(* CoDeSys 2.3.9.41 project: henkel.pro *)
(* Libraries: TcpIp.lib 21.3.13 07:03:14, TcBase.lib 14.5.09 12:14:08, TcSystem.lib 27.2.12 15:08:36, TcBaseMath.lib 27.7.04 12:07:56, TcMath.lib 23.9.04 15:15:30, TcMC2.lib 10.7.13 15:31:24, STANDARD.LIB 5.6.98 12:03:02, TcNC.lib 10.10.08 18:55:34, TcUtilities.lib 10.1.13 20:12:12, SysLibTargetVisu.lib 16.6.08 16:24:26, SysLibVisu.lib 7.7.04 18:17:22 *)

(* Task configuration *)
TASK Standard (PRIORITY := 1, INTERVAL := T#5ms);
	MAIN
END_TASK
TASK Fast (PRIORITY := 0, INTERVAL := T#1ms);
	MainFast();
END_TASK

(* Global variable list: Globale_Variablen *)
VAR_GLOBAL
	trigger1  AT %Q*: BOOL;			(*to tigger the auduino pin 6 motor running*)
	trigger2  AT %Q*: BOOL;			(*to tigger the auduino pin 7* in velocity*)
	encoderX:	ARRAY[1..5] OF		LREAL;
	encoderY:	ARRAY[1..5] OF		LREAL;
	heading:		ARRAY[1..5] OF		LREAL;
	reset:		BOOL;
	home: BOOL;
	combinedX: LREAL;
	combinedY: LREAL;
	combinedH: LREAL;
(*for ROS*)
	robotPosX:	LREAL;
	robotPosY:	LREAL;
	robotPosTheta:	LREAL;
	robotVelX:	LREAL;
	robotVelY:	LREAL;
	robotVelTheta:	LREAL;
(*
###################
	TwinCAT NC Achsen
###################
*)


	Axis1 : AXIS_REF;
	PowerAxis1: MC_Power;
	MoveAxis1: MC_MoveVelocity;
	MoveAxis12: MC_MoveVelocity;
	ResetAxis1: MC_Reset;		(* debug function block output data *)
	HaltAxis1: MC_Halt;

	Axis2 : AXIS_REF;
	PowerAxis2: MC_Power;
	MoveAxis2: MC_MoveVelocity;
	MoveAxis22: MC_MoveVelocity;
	ResetAxis2: MC_Reset;		(* debug function block output data *)
	HaltAxis2: MC_Halt;

	Axis3 : AXIS_REF;
	PowerAxis3: MC_Power;
	MoveAxis3: MC_MoveVelocity;
	MoveAxis32: MC_MoveVelocity;
	ResetAxis3: MC_Reset;		(* debug function block output data *)
	HaltAxis3: MC_Halt;

	Axis4 : AXIS_REF;
	PowerAxis4: MC_Power;
	MoveAxis4: MC_MoveVelocity;
	MoveAxis42: MC_MoveVelocity;
	ResetAxis4: MC_Reset;		(* debug function block output data *)
	HaltAxis4: MC_Halt;
END_VAR

(* Global variable list: TwinCAT_Configuration *)
(* Generated automatically by TwinCAT - (read only) *)
VAR_CONFIG
	MainFast.fblocalization.encoder1.PlcToNc AT %QB1156 : PLCTONC_AXIS_REF;
	MainFast.fblocalization.encoder1.NcToPlc AT %IB1152 : NCTOPLC_AXIS_REF;
	MainFast.fblocalization.encoder2.PlcToNc AT %QB1284 : PLCTONC_AXIS_REF;
	MainFast.fblocalization.encoder2.NcToPlc AT %IB1280 : NCTOPLC_AXIS_REF;
	MainFast.fblocalization.encoder3.PlcToNc AT %QB1412 : PLCTONC_AXIS_REF;
	MainFast.fblocalization.encoder3.NcToPlc AT %IB1408 : NCTOPLC_AXIS_REF;
	MainFast.fblocalization.encoder4.PlcToNc AT %QB1540 : PLCTONC_AXIS_REF;
	MainFast.fblocalization.encoder4.NcToPlc AT %IB1536 : NCTOPLC_AXIS_REF;
	.trigger1 AT %QX1152.0 : BOOL;
	.trigger2 AT %QX1152.1 : BOOL;
END_VAR

(* Global variable list: Variablen_Konfiguration *)
VAR_CONFIG
	Axis1.PlcToNc AT %QB128 : PLCTONC_AXIS_REF;	(*  ~ {LinkedWith:TINC^NC-Task 1 SAF^Achsen^Achse 1^Eingänge^Achse 1_FromPlc} *)
	Axis1.NcToPlc AT %IB128 : NCTOPLC_AXIS_REF;	(*  ~ {LinkedWith:TINC^NC-Task 1 SAF^Achsen^Achse 1^Ausgänge^Achse 1_ToPlc} *)
	Axis2.PlcToNc AT %QB256 : PLCTONC_AXIS_REF;	(*  ~ {LinkedWith:TINC^NC-Task 1 SAF^Achsen^Achse 2^Eingänge^Achse 2_FromPlc} *)
	Axis2.NcToPlc AT %IB256 : NCTOPLC_AXIS_REF;	(*  ~ {LinkedWith:TINC^NC-Task 1 SAF^Achsen^Achse 2^Ausgänge^Achse 2_ToPlc} *)
	Axis3.PlcToNc AT %QB512 : PLCTONC_AXIS_REF;
	Axis3.NcToPlc AT %IB512 : NCTOPLC_AXIS_REF;
	Axis4.PlcToNc AT %QB1024 : PLCTONC_AXIS_REF;
	Axis4.NcToPlc AT %IB1024 : NCTOPLC_AXIS_REF;
END_VAR

(* Data type *)
TYPE MoveState_NC :
(
	NC_INIT,
	NC_ENABLE,
	NC_MOVE,
	NC_MOVENEXT,
	NC_ERROR,
	NC_RESET
);
END_TYPE

(* POU MAIN, ST *)
PROGRAM MAIN
VAR
	fbPLC_Reset:  PLC_Reset;
	fbPLC_Start:  PLC_Start;
	state_NC : MoveState_NC;
(* manual runnning*)
	Manual: BOOL:=FALSE;
	bEnable: 			BOOL;										(* gibt die Achse frei *)
	bReset_Axis: 			BOOL;										(* Reset der Achse *)
	bAxis_Ready:		ARRAY[1..5] OF	BOOL;						(* Checks whether the axis is ready *)
	bMoveCombination:	ARRAY[1..10] OF		BOOL;					(*the combined movement*)
	i: INT;
	MotionReq: BOOL;
	timeToMove: TIME;
	directionToMove: INT;
	timeToMoveReal: LREAL;
	speedToMove:LREAL:=603;
	timeUp: BOOL;
	timerOn: BOOL;
	fbTON1: TON;



(*
###################
ROS TCP/IP CONNECTION
###################
*)
	myROS_connect_receiveData:				ROS_connect_receiveData;
	myROS_connect_sendData:				ROS_connect_sendData;
	myROS_disconnect:			ROS_disconnect;
	myROS_receiveData:			ROS_receiveData;
	myROS_sendData:			ROS_sendData;
	myROS_convertSendData:		ROS_convertSendData;

	ROS_tcpSocketReceiveData: T_HSOCKET;
	ROS_connectionOpenReceiveData: BOOL:=FALSE;

	ROS_tcpSocketSendData: T_HSOCKET;
	ROS_connectionOpenSendData: BOOL:=FALSE;

	ROS_closeConnection: BOOL:=TRUE;

	ROS_velAxis1: LREAL := 0;
	ROS_velAxis2: LREAL := 0;
	ROS_velAxis3: LREAL := 0;
	ROS_velAxis4: LREAL := 0;

	ROS_RobotPosX: LREAL := 0;
	ROS_RobotPosY: LREAL := 0;
	ROS_RobotPosTheta: LREAL:= 0;
	ROS_RobotVelX: LREAL:= 0;
	ROS_RobotVelY: LREAL:= 0;
	ROS_RobotVelTheta: LREAL:= 0;

	sendBufferREAL: LREAL:=0;
	sendBuffer: STRING;
	sendTakt: LREAL := 0;
	(*#END# ROS variables*)



	vel_last1 : LREAL;
	vel_current1 : LREAL;
	vel_last2 : LREAL;
	vel_current2 : LREAL;
	vel_last3 : LREAL;
	vel_current3 : LREAL;
	vel_last4 : LREAL;
	vel_current4 : LREAL;

(*
###################
ODOMETRY
###################
*)



	startTimer1: BOOL;
	timer1On: BOOL;

	firstStart: BOOL;
	Q: BOOL;
	startPLC: BOOL;
	oldSpeedX: LREAL;
	oldSpeedY: LREAL;
	oldSpeedH: LREAL;

(*JOSTICK*)
	connectJs:			jsConnect;
	disconnectJs:			jsDisconnect;
	receiveJsData:				jsReceiveData;
	tcpSockeJst: T_HSOCKET;
	connectionOpen_js: BOOL:=FALSE;
	closeConnection_js: BOOL:=TRUE;
	XAxis: LREAL;
	YAxis: LREAL;
	ZAxis: LREAL;
	botton: LREAL;

	myWP_tcpSocket: T_HSOCKET;
	myWP_connect:		WP_connect;
	myWP_disconnect:	WP_Disconnect;
	myWP_receiveData:	WP_ReceiveData;
	myWP_connected: BOOL := FALSE;
	myWP_connectionClosed: BOOL:=TRUE;
	wpBotton: LREAL;
END_VAR
(*
##
## This code was built by Theng Chua and Christian Scheifele, University of Stuttgart, 2014.
## It contains complete segments from Chris Jarrett, Auckland University, 2014
## and is derived in part from the TCP/IP server example on www.beckhoff.com
##
*)

(*
###################
Manual
###################
*)
IF (Manual=TRUE) THEN
	IF (reset=TRUE) THEN
	trigger1:=FALSE;
	trigger2:=TRUE;
	fbPLC_Reset(port:=801,RESET:=TRUE);
	fbPLC_Start(port:=801,start:=TRUE);
	reset:=FALSE;
	trigger1:=FALSE;
	trigger2:=FALSE;
	END_IF

	FOR i:=1 TO 10 BY 1 DO
		IF(bMoveCombination[i]) THEN
			directionToMove:=i;
			MotionReq:=TRUE;
		END_IF
	END_FOR

	IF(MotionReq=TRUE) THEN
		CASE directionToMove OF
		1:	ROS_velAxis1:= -speedToMove;
			ROS_velAxis2:= 0;
			ROS_velAxis3:= 0;
			ROS_velAxis4:= -speedToMove;
		2:	ROS_velAxis1:= -speedToMove;
			ROS_velAxis2:= -speedToMove;
			ROS_velAxis3:= -speedToMove;
			ROS_velAxis4:= -speedToMove;
		3:	ROS_velAxis1:= 0;
			ROS_velAxis2:= -speedToMove;
			ROS_velAxis3:= -speedToMove;
			ROS_velAxis4:= 0;
		4:	ROS_velAxis1:= -speedToMove;
			ROS_velAxis2:= speedToMove;
			ROS_velAxis3:= speedToMove;
			ROS_velAxis4:= -speedToMove;
		5:	ROS_velAxis1:= speedToMove;
			ROS_velAxis2:= -speedToMove;
			ROS_velAxis3:= -speedToMove;
			ROS_velAxis4:= speedToMove;
		6:	ROS_velAxis1:= 0;
			ROS_velAxis2:= speedToMove;
			ROS_velAxis3:= speedToMove;
			ROS_velAxis4:= 0;
		7:	ROS_velAxis1:= speedToMove;
			ROS_velAxis2:= speedToMove;
			ROS_velAxis3:= speedToMove;
			ROS_velAxis4:= speedToMove;
		8:	ROS_velAxis1:= speedToMove;
			ROS_velAxis2:= 0;
			ROS_velAxis3:= 0;
			ROS_velAxis4:= speedToMove;
		9:	ROS_velAxis1:= -speedToMove;
			ROS_velAxis2:= speedToMove;
			ROS_velAxis3:= -speedToMove;
			ROS_velAxis4:= speedToMove;
		10:	ROS_velAxis1:= speedToMove;
			ROS_velAxis2:= -speedToMove;
			ROS_velAxis3:= speedToMove;
			ROS_velAxis4:= -speedToMove;
		ELSE
			ROS_velAxis1:= 0;
			ROS_velAxis2:= 0;
			ROS_velAxis3:= 0;
			ROS_velAxis4:= 0;
		END_CASE
	timetomove:= REAL_TO_TIME (timeToMoveReal);
	timerOn:=TRUE;
	END_IF

	fbTON1(IN:=timerOn, PT:=timeToMove, Q=>timeUp, ET=>);

	IF (timeUp=TRUE)  THEN
	MotionReq:=FALSE;
	bMoveCombination[directionToMove]:=FALSE;
	ROS_velAxis1:= 0;
	ROS_velAxis2:= 0;
	ROS_velAxis3:= 0;
	ROS_velAxis4:= 0;
	directionToMove:=0;
	timerOn:=FALSE;
	END_IF
(*
###################
ODOMETRY
###################
*)

	IF (vel_current1<>0 OR vel_current2<>0 OR vel_current3<>0 OR vel_current4<>0) THEN trigger1:=TRUE;
	ELSE trigger1:=FALSE;
	END_IF

	trigger2:=(MoveAxis1.InVelocity AND MoveAxis2.InVelocity AND MoveAxis3.InVelocity AND MoveAxis4.InVelocity) OR (MoveAxis12.InVelocity AND MoveAxis22.InVelocity AND MoveAxis32.InVelocity AND MoveAxis42.InVelocity);

ELSE
(*
###################
ROS TCP/IP CONNECTION
###################

Close TCP port from last time-remove after DEBUG
	
		IF ROS_closeConnection THEN
		myROS_disconnect(bCloseAll:=ROS_closeConnection);
		ROS_closeConnection:=FALSE;
		END_IF*)

		(*Open a connection to ROS - Receive Data*)
		IF NOT ROS_connectionOpenReceiveData THEN
		myROS_connect_receiveData(RosConnected=>ROS_connectionOpenReceiveData, socketToUse=>ROS_tcpSocketReceiveData);
		END_IF
		IF ROS_connectionOpenReceiveData THEN
		myROS_receiveData(socketToUse:=ROS_tcpSocketReceiveData,velAxis1=>ROS_velAxis1, velAxis2=>ROS_velAxis2, velAxis3=>ROS_velAxis3, velAxis4=>ROS_velAxis4);
		END_IF

		(*Open a connection to ROS - Send Data*)
		IF NOT ROS_connectionOpenSendData THEN
		myROS_connect_sendData(RosConnected=>ROS_connectionOpenSendData, socketToUse=>ROS_tcpSocketSendData);
		END_IF

		(*ODOMETRY SORCE*)
		ROS_RobotPosX := robotPosY;
		ROS_RobotPosY := robotPosX;
		ROS_RobotPosTheta := robotPosTheta;
		ROS_RobotVelX := RobotVelY;
		ROS_RobotVelY := RobotVelX;
		ROS_RobotVelTheta := RobotVelTheta;

		IF ROS_connectionOpenSendData THEN
		(* TAKTZEIT EINSTELLEN *)
		sendTakt := sendTakt + 0.1;
			IF sendTakt > 1THEN
			myROS_convertSendData(robotPosX:=ROS_RobotPosX, robotPosY:=ROS_RobotPosY, robotPosTheta:= ROS_RobotPosTheta, robotVelX:=ROS_RobotVelX, robotVelY:=ROS_RobotVelY, robotVelTheta:=ROS_RobotVelTheta, send_message=>sendBuffer );
			myROS_sendData(sendBuffer:=sendBuffer, socketToUse:=ROS_tcpSocketSendData);
			sendTakt := 0;
			END_IF
		END_IF



	(*JOSTICK*)
	(*Close TCP port from last time-remove after DEBUG*)
	IF closeConnection_js THEN
	disconnectJs(bCloseAll:=closeConnection_js);
	closeConnection_js:=FALSE;
	END_IF

	(*Open a connection*)
	IF (connectionOpen_js=FALSE) THEN
	connectJs(arduinoConnected=>connectionOpen_js, socketToUse=>tcpSockeJst);
	END_IF

	IF (connectionOpen_js=TRUE) THEN
	receiveJsData(socketToUse:=tcpSockeJst ,botton=>botton, xAxis=>XAxis, yAxis=>YAxis, zAxis=>ZAxis);
	END_IF

	(*IF  (botton = 48 OR botton = 32) THEN
	ROS_velAxis1:= -YAxis+XAxis-ZAxis;
	ROS_velAxis2:= -YAxis-XAxis+ZAxis;
	ROS_velAxis3:= -YAxis-XAxis-ZAxis;
	ROS_velAxis4:= -YAxis+XAxis+ZAxis;
	ELSE
	ROS_velAxis1:= 0;
	ROS_velAxis2:= 0;
	ROS_velAxis3:= 0;
	ROS_velAxis4:= 0;
	END_IF*)

(*Windows Phone Connection*)

	IF (myWP_connectionClosed) THEN
	myWP_disconnect(bCloseAll:=myWP_connectionClosed);
	myWP_connectionClosed:=FALSE;
	END_IF

	IF (myWP_connected=FALSE) THEN
	myWP_connect(WPConnected=>myWP_connected, socketToUse=>myWP_tcpSocket);
	END_IF

	IF (myWP_connected=TRUE) THEN
	myWP_receiveData(socketToUse:=myWP_tcpSocket ,botton=>wpBotton, xAxis=>XAxis, yAxis=>YAxis, zAxis=>ZAxis);
		(*IF(wpBotton <> 0 ) THEN
			ROS_velAxis1:= -YAxis+XAxis-ZAxis;
			ROS_velAxis2:= -YAxis-XAxis+ZAxis;
			ROS_velAxis3:= -YAxis-XAxis-ZAxis;
			ROS_velAxis4:= -YAxis+XAxis+ZAxis;
		END_IF*)
		wpBotton := 0;
	END_IF

END_IF (* for manual running*)

(*
###################
TwinCAT NC Achsen
###################
*)
Axis1.ReadStatus;
Axis2.ReadStatus;
Axis3.ReadStatus;
Axis4.ReadStatus;

vel_current1 := -ROS_velAxis1;
vel_current2 := ROS_velAxis2;
vel_current3 := -ROS_velAxis3;
vel_current4 := ROS_velAxis4;

(* move axis using a state machine *)
CASE state_NC OF
		NC_INIT :	(* initialisation *)
			(* initialize all function blocks *)
			MoveAxis1.Execute := FALSE;
			ResetAxis1.Execute := FALSE;
			MoveAxis2.Execute := FALSE;
			ResetAxis2.Execute := FALSE;
			MoveAxis3.Execute := FALSE;
			ResetAxis3.Execute := FALSE;
			MoveAxis4.Execute := FALSE;
			ResetAxis4.Execute := FALSE;
			MoveAxis12.Execute := FALSE;
			MoveAxis22.Execute := FALSE;
			MoveAxis32.Execute := FALSE;
			MoveAxis42.Execute := FALSE;
			HaltAxis1.Execute := FALSE;
			HaltAxis2.Execute := FALSE;
			HaltAxis3.Execute := FALSE;
			HaltAxis4.Execute := FALSE;

			state_NC := NC_ENABLE;

		NC_ENABLE :
			PowerAxis1.Enable := TRUE;
			PowerAxis1.Enable_Positive := TRUE;
			PowerAxis1.Enable_Negative := TRUE;
			PowerAxis2.Enable := TRUE;
			PowerAxis2.Enable_Positive := TRUE;
			PowerAxis2.Enable_Negative := TRUE;
			PowerAxis3.Enable := TRUE;
			PowerAxis3.Enable_Positive := TRUE;
			PowerAxis3.Enable_Negative := TRUE;
			PowerAxis4.Enable := TRUE;
			PowerAxis4.Enable_Positive := TRUE;
			PowerAxis4.Enable_Negative := TRUE;

			IF PowerAxis1.Status AND PowerAxis2.Status AND PowerAxis3.Status AND PowerAxis4.Status THEN
				state_NC := NC_MOVE;
			ELSIF PowerAxis1.Error AND PowerAxis2.Error AND PowerAxis3.Error AND PowerAxis4.Error THEN
				state_NC := NC_ERROR;
			END_IF

		NC_MOVE :
			IF vel_current1>0 THEN
				HaltAxis1.Execute := FALSE;
				MoveAxis1.Direction := MC_Positive_Direction;
				MoveAxis1.Velocity := vel_current1;
				MoveAxis1.BufferMode := MC_Aborting;
				MoveAxis1.Execute := TRUE;
			ELSIF vel_current1<0 THEN
				HaltAxis1.Execute := FALSE;
				MoveAxis1.Direction := MC_Negative_Direction;
				MoveAxis1.Velocity := -vel_current1;
				MoveAxis1.BufferMode := MC_Aborting;
				MoveAxis1.Execute := TRUE;
			ELSE
				HaltAxis1.BufferMode := MC_Aborting;
				HaltAxis1.Execute := TRUE;
			END_IF;


			IF vel_current2>0 THEN
				HaltAxis2.Execute := FALSE;
				MoveAxis2.Direction := MC_Positive_Direction;
				MoveAxis2.Velocity := vel_current2;
				MoveAxis2.BufferMode := MC_Aborting;
				MoveAxis2.Execute := TRUE;
			ELSIF vel_current2<0 THEN
				HaltAxis2.Execute := FALSE;
				MoveAxis2.Direction := MC_Negative_Direction;
				MoveAxis2.Velocity := -vel_current2;
				MoveAxis2.BufferMode := MC_Aborting;
				MoveAxis2.Execute := TRUE;
			ELSE
				HaltAxis2.BufferMode := MC_Aborting;
				HaltAxis2.Execute := TRUE;
			END_IF;


			IF vel_current3>0 THEN
				HaltAxis3.Execute := FALSE;
				MoveAxis3.Direction := MC_Positive_Direction;
				MoveAxis3.Velocity := vel_current3;
				MoveAxis3.BufferMode := MC_Aborting;
				MoveAxis3.Execute := TRUE;
			ELSIF vel_current3<0 THEN
				HaltAxis3.Execute := FALSE;
				MoveAxis3.Direction := MC_Negative_Direction;
				MoveAxis3.Velocity := -vel_current3;
				MoveAxis3.BufferMode := MC_Aborting;
				MoveAxis3.Execute := TRUE;
			ELSE
				HaltAxis3.BufferMode := MC_Aborting;
				HaltAxis3.Execute := TRUE;
			END_IF;


			IF vel_current4>0 THEN
				HaltAxis4.Execute := FALSE;
				MoveAxis4.Direction := MC_Positive_Direction;
				MoveAxis4.Velocity := vel_current4;
				MoveAxis4.BufferMode := MC_Aborting;
				MoveAxis4.Execute := TRUE;
			ELSIF vel_current4<0 THEN
				HaltAxis4.Execute := FALSE;
				MoveAxis4.Direction := MC_Negative_Direction;
				MoveAxis4.Velocity := -vel_current4;
				MoveAxis4.BufferMode := MC_Aborting;
				MoveAxis4.Execute := TRUE;
			ELSE
				HaltAxis4.BufferMode := MC_Aborting;
				HaltAxis4.Execute := TRUE;
			END_IF;

			IF vel_last1<>vel_current1 OR vel_last2<>vel_current2 OR vel_last3<>vel_current3 OR vel_last4<>vel_current4 THEN
				MoveAxis1.Execute := FALSE;
				MoveAxis2.Execute := FALSE;
				MoveAxis3.Execute := FALSE;
				MoveAxis4.Execute := FALSE;
				vel_last1 := vel_current1;
				vel_last2 := vel_current2;
				vel_last3 := vel_current3;
				vel_last4 := vel_current4;
				state_NC := NC_MOVENEXT;
			END_IF;
			IF  MoveAxis1.CommandAborted OR MoveAxis1.Error OR MoveAxis2.CommandAborted OR MoveAxis2.Error OR MoveAxis3.CommandAborted OR MoveAxis3.Error OR MoveAxis4.CommandAborted OR MoveAxis4.Error THEN
				state_NC := NC_MOVE;
			END_IF

		NC_MOVENEXT :
			IF vel_current1>0 THEN
				HaltAxis1.Execute := FALSE;
				MoveAxis12.Direction := MC_Positive_Direction;
				MoveAxis12.Velocity := vel_current1;
				MoveAxis12.BufferMode := MC_Aborting;
				MoveAxis12.Execute := TRUE;
			ELSIF vel_current1<0 THEN
				HaltAxis1.Execute := FALSE;
				MoveAxis12.Direction := MC_Negative_Direction;
				MoveAxis12.Velocity := -vel_current1;
				MoveAxis12.BufferMode := MC_Aborting;
				MoveAxis12.Execute := TRUE;
			ELSE
				HaltAxis1.BufferMode := MC_Aborting;
				HaltAxis1.Execute := TRUE;
			END_IF;


			IF vel_current2>0 THEN
				HaltAxis2.Execute := FALSE;
				MoveAxis22.Direction := MC_Positive_Direction;
				MoveAxis22.Velocity := vel_current2;
				MoveAxis22.BufferMode := MC_Aborting;
				MoveAxis22.Execute := TRUE;
			ELSIF vel_current2<0 THEN
				HaltAxis2.Execute := FALSE;
				MoveAxis22.Direction := MC_Negative_Direction;
				MoveAxis22.Velocity := -vel_current2;
				MoveAxis22.BufferMode := MC_Aborting;
				MoveAxis22.Execute := TRUE;
			ELSE
				HaltAxis2.BufferMode := MC_Aborting;
				HaltAxis2.Execute := TRUE;
			END_IF;


			IF vel_current3>0 THEN
				HaltAxis3.Execute := FALSE;
				MoveAxis32.Direction := MC_Positive_Direction;
				MoveAxis32.Velocity := vel_current3;
				MoveAxis32.BufferMode := MC_Aborting;
				MoveAxis32.Execute := TRUE;
			ELSIF vel_current3<0 THEN
				HaltAxis3.Execute := FALSE;
				MoveAxis32.Direction := MC_Negative_Direction;
				MoveAxis32.Velocity := -vel_current3;
				MoveAxis32.BufferMode := MC_Aborting;
				MoveAxis32.Execute := TRUE;
			ELSE
				HaltAxis3.BufferMode := MC_Aborting;
				HaltAxis3.Execute := TRUE;
			END_IF;


			IF vel_current4>0 THEN
				HaltAxis4.Execute := FALSE;
				MoveAxis42.Direction := MC_Positive_Direction;
				MoveAxis42.Velocity := vel_current4;
				MoveAxis42.BufferMode := MC_Aborting;
				MoveAxis42.Execute := TRUE;
			ELSIF vel_current4<0 THEN
				HaltAxis4.Execute := FALSE;
				MoveAxis42.Direction := MC_Negative_Direction;
				MoveAxis42.Velocity := -vel_current4;
				MoveAxis42.BufferMode := MC_Aborting;
				MoveAxis42.Execute := TRUE;
			ELSE
				HaltAxis4.BufferMode := MC_Aborting;
				HaltAxis4.Execute := TRUE;
			END_IF;

			IF vel_last1<>vel_current1 OR vel_last2<>vel_current2 OR vel_last3<>vel_current3 OR vel_last4<>vel_current4 THEN
				MoveAxis12.Execute := FALSE;
				MoveAxis22.Execute := FALSE;
				MoveAxis32.Execute := FALSE;
				MoveAxis42.Execute := FALSE;
				vel_last1 := vel_current1;
				vel_last2 := vel_current2;
				vel_last3 := vel_current3;
				vel_last4 := vel_current4;
				state_NC := NC_MOVE;
			END_IF;
			IF  MoveAxis12.CommandAborted OR MoveAxis12.Error OR MoveAxis22.CommandAborted OR MoveAxis22.Error OR MoveAxis32.CommandAborted OR MoveAxis32.Error OR MoveAxis42.CommandAborted OR MoveAxis42.Error THEN
				state_NC := NC_MOVE;
			END_IF


		NC_ERROR :
			IF Axis1.Status.Error OR Axis2.Status.Error OR Axis3.Status.Error OR Axis4.Status.Error THEN
				state_NC := NC_RESET;	(* axis error requires reset *)
			ELSE
				state_NC := NC_INIT;		(* function block errors don't need a reset *)
			END_IF

		NC_RESET :
			ResetAxis1.Execute := TRUE;
			ResetAxis2.Execute := TRUE;
			ResetAxis3.Execute := TRUE;
			ResetAxis4.Execute := TRUE;
			IF ResetAxis1.Done AND ResetAxis2.Done AND ResetAxis3.Done AND ResetAxis4.Done THEN
				state_NC := NC_INIT;
			ELSIF ResetAxis1.Error OR ResetAxis2.Error OR ResetAxis3.Error OR ResetAxis4.Error THEN
				state_NC := NC_INIT; (* can't do anything here *)
			END_IF

END_CASE

ActPower;	(* call the power function block *)
ActMove;	(* call the move function block *)
ActReset;	(* call the reset function block *)
ActHaltAxis1;
ActHaltAxis2;
ActHaltAxis3;
ActHaltAxis4;
END_PROGRAM
ACTION ActHaltAxis1:
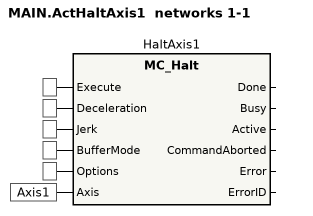
_FBD_ (* Function Block Diagram *)
NETWORK 1
	HaltAxis1:MC_Halt(Execute: , Deceleration: , Jerk: , BufferMode: , Options: , Axis: Axis1)
_END_FBD_
END_ACTION
ACTION ActHaltAxis2:
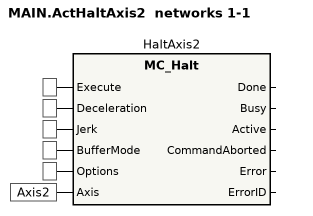
_FBD_ (* Function Block Diagram *)
NETWORK 1
	HaltAxis2:MC_Halt(Execute: , Deceleration: , Jerk: , BufferMode: , Options: , Axis: Axis2)
_END_FBD_
END_ACTION
ACTION ActHaltAxis3:
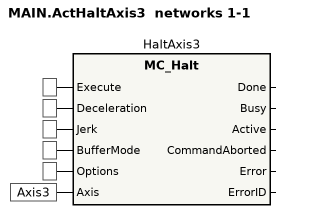
_FBD_ (* Function Block Diagram *)
NETWORK 1
	HaltAxis3:MC_Halt(Execute: , Deceleration: , Jerk: , BufferMode: , Options: , Axis: Axis3)
_END_FBD_
END_ACTION
ACTION ActHaltAxis4:
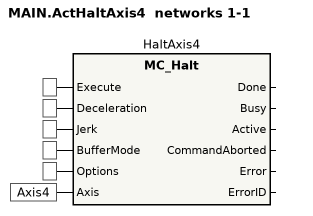
_FBD_ (* Function Block Diagram *)
NETWORK 1
	HaltAxis4:MC_Halt(Execute: , Deceleration: , Jerk: , BufferMode: , Options: , Axis: Axis4)
_END_FBD_
END_ACTION
ACTION ActMove:
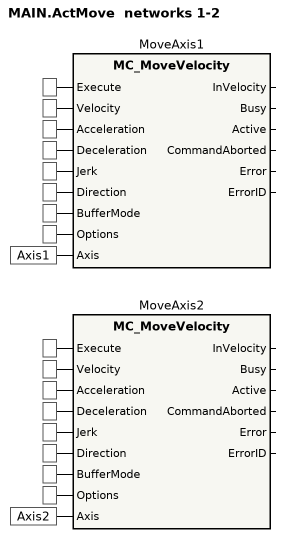
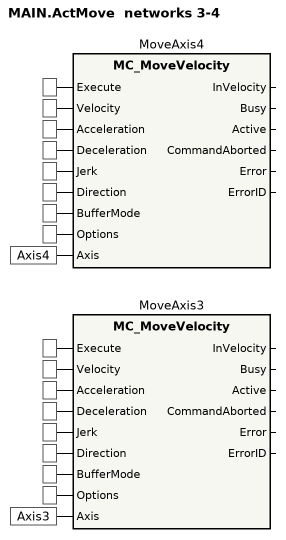
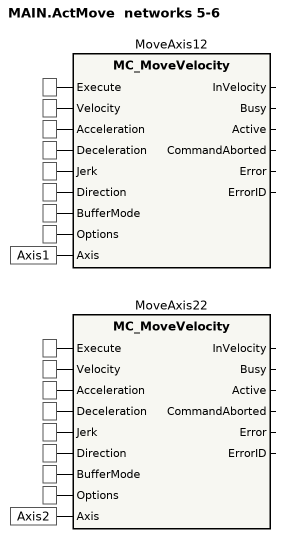
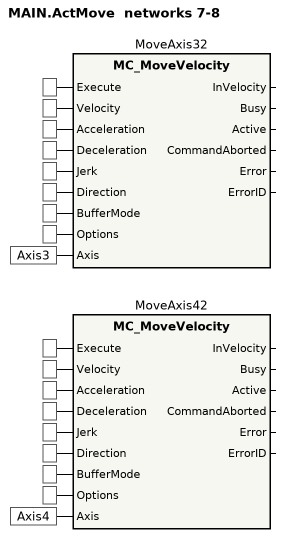
_FBD_ (* Function Block Diagram *)
NETWORK 1
	MoveAxis1:MC_MoveVelocity(Execute: , Velocity: , Acceleration: , Deceleration: , Jerk: , Direction: , BufferMode: , Options: , Axis: Axis1)
NETWORK 2
	MoveAxis2:MC_MoveVelocity(Execute: , Velocity: , Acceleration: , Deceleration: , Jerk: , Direction: , BufferMode: , Options: , Axis: Axis2)
NETWORK 3
	MoveAxis4:MC_MoveVelocity(Execute: , Velocity: , Acceleration: , Deceleration: , Jerk: , Direction: , BufferMode: , Options: , Axis: Axis4)
NETWORK 4
	MoveAxis3:MC_MoveVelocity(Execute: , Velocity: , Acceleration: , Deceleration: , Jerk: , Direction: , BufferMode: , Options: , Axis: Axis3)
NETWORK 5
	MoveAxis12:MC_MoveVelocity(Execute: , Velocity: , Acceleration: , Deceleration: , Jerk: , Direction: , BufferMode: , Options: , Axis: Axis1)
NETWORK 6
	MoveAxis22:MC_MoveVelocity(Execute: , Velocity: , Acceleration: , Deceleration: , Jerk: , Direction: , BufferMode: , Options: , Axis: Axis2)
NETWORK 7
	MoveAxis32:MC_MoveVelocity(Execute: , Velocity: , Acceleration: , Deceleration: , Jerk: , Direction: , BufferMode: , Options: , Axis: Axis3)
NETWORK 8
	MoveAxis42:MC_MoveVelocity(Execute: , Velocity: , Acceleration: , Deceleration: , Jerk: , Direction: , BufferMode: , Options: , Axis: Axis4)
_END_FBD_
END_ACTION
ACTION ActPower:
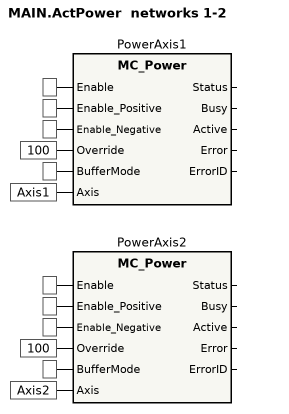
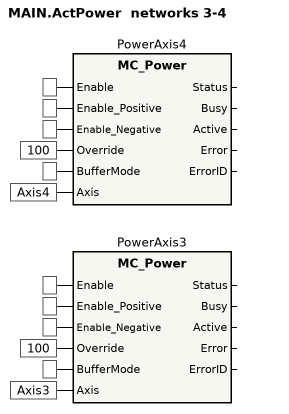
_FBD_ (* Function Block Diagram *)
NETWORK 1
	PowerAxis1:MC_Power(Enable: , Enable_Positive: , Enable_Negative: , Override: 100, BufferMode: , Axis: Axis1)
NETWORK 2
	PowerAxis2:MC_Power(Enable: , Enable_Positive: , Enable_Negative: , Override: 100, BufferMode: , Axis: Axis2)
NETWORK 3
	PowerAxis4:MC_Power(Enable: , Enable_Positive: , Enable_Negative: , Override: 100, BufferMode: , Axis: Axis4)
NETWORK 4
	PowerAxis3:MC_Power(Enable: , Enable_Positive: , Enable_Negative: , Override: 100, BufferMode: , Axis: Axis3)
_END_FBD_
END_ACTION
ACTION ActReset:
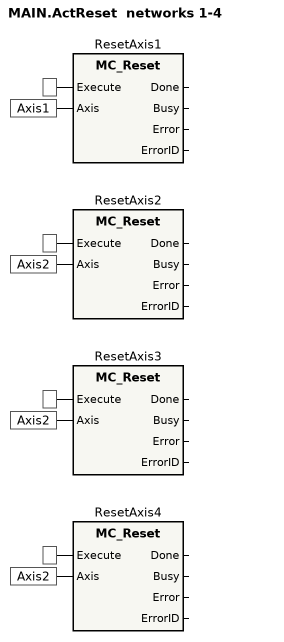
_FBD_ (* Function Block Diagram *)
NETWORK 1
	ResetAxis1:MC_Reset(Execute: , Axis: Axis1)
NETWORK 2
	ResetAxis2:MC_Reset(Execute: , Axis: Axis2)
NETWORK 3
	ResetAxis3:MC_Reset(Execute: , Axis: Axis2)
NETWORK 4
	ResetAxis4:MC_Reset(Execute: , Axis: Axis2)
_END_FBD_
END_ACTION

(* POU ROS_connect_receiveData, ST *)
FUNCTION_BLOCK ROS_connect_receiveData
VAR


	(*Functions*)
	openSocket: BOOL:=FALSE;
	fb_listen: FB_SocketListen;
	fb_accept: FB_SocketAccept;
	(*Timers*)
	fbAcceptTON: TON;

	(*TCP socket variables*)
	activeSocketHandle: T_HSOCKET;
	socketHandle: T_HSOCKET;



	(*Error variables*)
	listenError: UDINT:=0;
	acceptError: UDINT;
	listenErrSet: BOOL;
	closeError: UDINT;
	sendError: UDINT;
	receiveError: UDINT;
	bSendError: BOOL;


	(*Trigger Variables*)
	bCloseAll: BOOL := TRUE;

	(*Connection information*)
	portNumber: INT:=711;
	bAccepted: BOOL;

	(*Constants*)
	PLCPRJ_ACCEPT_POLLING_TIME: TIME:=T#1s;

	display: LREAL;
	heading: LREAL;

	state: INT:=0;

	xDist: LREAL;
	yDist: LREAL;
	zDist: LREAL;


	listening: BOOL;
END_VAR
VAR_OUTPUT
	RosConnected: BOOL;
	socketToUse: T_HSOCKET;
END_VAR
(*
##
## This code was built by Christian Scheifele, University of Stuttgart, 2014.
## It contains complete segments from Chris Jarrett, Auckland University, 2014
## and is derived in part from the TCP/IP server example on www.beckhoff.com
##
*)

CASE state OF
0:

IF(fb_Listen.hListener.localAddr.nPort=portNumber) THEN
RETURN;

ELSE
state:=1;
END_IF

1:
fb_listen
(
	sSrvNetId:='' ,
	sLocalHost:='',
	nLocalPort:=portNumber,
	bExecute:=TRUE,
	tTimeout:=T#5s,
	hListener=>socketHandle,
	nErrId=>listenError,
	bError=>listenErrSet,

);

	IF(fb_Listen.hListener.localAddr.nPort=portNumber) THEN
		fb_listen(bExecute:=FALSE); 		(*Start listening and move to the accept state*)

		state:=2;
	ELSE
		(*Return to the listening state*)
		state:=1;
	END_IF



2:

(*Start accepting a client connection*)
fbAcceptTON( IN := TRUE, PT := T#2s);  (*Start a timer to poll for the accepted connection*)
		IF fbAcceptTON.Q THEN
			fbAcceptTON( IN := FALSE );	(*Reset timer*)
			fb_accept(  bExecute := FALSE  ); (*Generate a rising edge to activate the accept function*)
			fb_accept(hListener := socketHandle, bExecute:= TRUE, hSocket=>activeSocketHandle );
			state:=3; (*Move to the state where the client is accepted*)

			fbAcceptTON( IN := FALSE);

		END_IF
3:
(*Complete accpeting the client connection*)
	fb_accept( bExecute := FALSE ); (*Reset the accept function to try connection again if necessary*)
	IF NOT fb_accept.bBusy THEN
		IF NOT fb_accept.bError THEN
			IF fb_accept.bAccepted THEN
				bAccepted := TRUE; (*If the client connection is accepted without error then move to the send state*)
				fb_accept(bExecute:=FALSE);
				socketToUse:=fb_accept.hSocket;
				state:=4;
			ELSE
				fb_listen(bExecute:=FALSE);
				fb_accept(bExecute:=FALSE);
				RosConnected:=FALSE; (*If the connection attempt was not successful, return the boolean as false*)
				fbAcceptTON( IN := FALSE);
				state:=2;
			END_IF
		END_IF
	END_IF
4:
RosConnected:=TRUE;
RETURN;

END_CASE;
END_FUNCTION_BLOCK

(* POU ROS_connect_sendData, ST *)
FUNCTION_BLOCK ROS_connect_sendData
VAR


	(*Functions*)
	openSocket: BOOL:=FALSE;
	fb_listen: FB_SocketListen;
	fb_accept: FB_SocketAccept;
	(*Timers*)
	fbAcceptTON: TON;

	(*TCP socket variables*)
	activeSocketHandle: T_HSOCKET;
	socketHandle: T_HSOCKET;



	(*Error variables*)
	listenError: UDINT:=0;
	acceptError: UDINT;
	listenErrSet: BOOL;
	closeError: UDINT;
	sendError: UDINT;
	receiveError: UDINT;
	bSendError: BOOL;


	(*Trigger Variables*)
	bCloseAll: BOOL := TRUE;

	(*Connection information*)
	portNumber: INT:=712;
	bAccepted: BOOL;

	(*Constants*)
	PLCPRJ_ACCEPT_POLLING_TIME: TIME:=T#1s;

	display: LREAL;
	heading: LREAL;

	state: INT:=0;

	xDist: LREAL;
	yDist: LREAL;
	zDist: LREAL;


	listening: BOOL;
END_VAR
VAR_OUTPUT
	RosConnected: BOOL;
	socketToUse: T_HSOCKET;
END_VAR
(*
##
## This code was built by Christian Scheifele, University of Stuttgart, 2014.
## It contains complete segments from Chris Jarrett, Auckland University, 2014
## and is derived in part from the TCP/IP server example on www.beckhoff.com
##
*)

CASE state OF
0:

IF(fb_Listen.hListener.localAddr.nPort=portNumber) THEN
RETURN;

ELSE
state:=1;
END_IF

1:
(*This code was built by Chris Jarrett, Auckland University, 2014. It is derived in part from the TCP/IP server example on www.beckhoff.com*)
fb_listen
(
	sSrvNetId:='' ,
	sLocalHost:='',
	nLocalPort:=portNumber,
	bExecute:=TRUE,
	tTimeout:=T#5s,
	hListener=>socketHandle,
	nErrId=>listenError,
	bError=>listenErrSet,

);

	IF(fb_Listen.hListener.localAddr.nPort=portNumber) THEN
		fb_listen(bExecute:=FALSE); 		(*Start listening and move to the accept state*)

		state:=2;
	ELSE
		(*Return to the listening state*)
		state:=1;
	END_IF



2:

(*Start accepting a client connection*)
fbAcceptTON( IN := TRUE, PT := T#2s);  (*Start a timer to poll for the accepted connection*)
		IF fbAcceptTON.Q THEN
			fbAcceptTON( IN := FALSE );	(*Reset timer*)
			fb_accept(  bExecute := FALSE  ); (*Generate a rising edge to activate the accept function*)
			fb_accept(hListener := socketHandle, bExecute:= TRUE, hSocket=>activeSocketHandle );
			state:=3; (*Move to the state where the client is accepted*)

			fbAcceptTON( IN := FALSE);

		END_IF
3:
(*Complete accpeting the client connection*)
	fb_accept( bExecute := FALSE ); (*Reset the accept function to try connection again if necessary*)
	IF NOT fb_accept.bBusy THEN
		IF NOT fb_accept.bError THEN
			IF fb_accept.bAccepted THEN
				bAccepted := TRUE; (*If the client connection is accepted without error then move to the send state*)
				fb_accept(bExecute:=FALSE);
				socketToUse:=fb_accept.hSocket;
				state:=4;
			ELSE
				fb_listen(bExecute:=FALSE);
				fb_accept(bExecute:=FALSE);
				RosConnected:=FALSE; (*If the connection attempt was not successful, return the boolean as false*)
				fbAcceptTON( IN := FALSE);
				state:=2;
			END_IF
		END_IF
	END_IF
4:
RosConnected:=TRUE;
RETURN;

END_CASE;
END_FUNCTION_BLOCK

(* POU ROS_disconnect, ST *)
FUNCTION_BLOCK ROS_disconnect
VAR_INPUT
	bCloseAll: BOOL;
END_VAR
VAR_OUTPUT
	connectionClosed: BOOL;
END_VAR
VAR
	fb_closeAll: FB_SocketCloseAll;
END_VAR
(*
##
## This code was built by Christian Scheifele, University of Stuttgart, 2014.
## It contains complete segments from Chris Jarrett, Auckland University, 2014
## and is derived in part from the TCP/IP server example on www.beckhoff.com
##
*)


(*This function closes the TCP/IP port being used the ROS connection*)

IF bCloseAll THEN
	bCloseAll:=FALSE;
	(*Close all open ports*)
	fb_closeAll(sSrvNetId:='', bExecute:=TRUE, tTimeOut:=T#5s );
ELSE
	fb_closeAll(bExecute:=FALSE);
END_IF


(*Move to the listening state*)
IF NOT fb_closeAll.bError THEN
	connectionClosed:=TRUE;


ELSE
connectionClosed:=FALSE;
END_IF
RETURN;
END_FUNCTION_BLOCK

(* POU ROS_receiveData, ST *)
FUNCTION_BLOCK ROS_receiveData
VAR_INPUT
	socketToUse: T_HSOCKET;
END_VAR
VAR_OUTPUT
	dataReceived: BOOL;
	velAxis1: LREAL;
	velAxis2: LREAL;
	velAxis3: LREAL;
	velAxis4: LREAL;
END_VAR
VAR
	(*Connection timers*)
	fbReceiveTON: TON;
	fbResetTON:TON;
	reset: BOOL;
	timeup:BOOL;

 	(*Functions*)
	fb_receive: FB_SocketReceive;

	(*Send and receive data and variables*)
	receiveBuffer: ARRAY[0..27] OF BYTE;
	bytesReceived: UDINT;
	sendBuffer: STRING;
	sendBufferAddress: DWORD;
	cbReceived, startPos, endPos, idx : UDINT;
	cbFrame: UDINT;
	sFromClient: T_MaxString;
	overflow: BOOL;
	endFound: BOOL;

	(*Error variables*)
	acceptError: UDINT;
	receiveError: UDINT;

	state: INT:=1;
END_VAR
(*
##
## This code was built by Christian Scheifele, University of Stuttgart, 2014.
## It contains complete segments from Chris Jarrett, Auckland University, 2014
## and is derived in part from the TCP/IP server example on www.beckhoff.com
##
*)

CASE state OF
1:
(*Receive information*)
	fbReceiveTON(  IN := FALSE, PT:=T#0s); (*Receive first request immediately*)
	fbReceiveTON(  IN := TRUE ); (*Start a timer to ensure complete transfer of information*)

		IF fbReceiveTON.Q THEN
			fbReceiveTON(  IN := FALSE);
			fb_receive(bExecute:=FALSE);  (*Generate a rising edge to start receiving data*)
			fb_receive
			(
				sSrvNetId:='',
				hSocket :=socketToUse,
				cbLen:=SIZEOF(receiveBuffer)-cbReceived,
				pDest:=ADR(receiveBuffer)+cbReceived,
				tTimeout:=T#5s,
				nRecBytes=>bytesReceived,
				nErrId=>receiveError,
				bExecute:=TRUE,
			);

	(*Move to the receive completion state*)
	state:=2;
	END_IF

2:
(*Continue receiving data*)
	fb_receive( bExecute := FALSE );
	IF NOT fb_receive.bBusy THEN
		IF NOT fb_receive.bError THEN (*If no error has occurred then start the actual receiving of data*)

			IF (fb_receive.nRecBytes>0) THEN (*Bytes have been received*)

				startPos:=cbReceived; (*index of first data byte*)
				endPos:=cbReceived+fb_receive.nRecBytes-1; (*index of last byte*)
				cbReceived:=cbReceived+fb_receive.nRecBytes; (*Calculating the number of received data bytes*)
				cbFrame:=0; (*Reset the frame length*)


				IF cbReceived<SIZEOF(sFromClient) THEN (*no overflow*)
					fbReceiveTON(IN:=FALSE, PT:=T#0S);

					(*Search for the string delimiter(separation character for different strings)*)
					FOR idx:=startPos TO endPos BY 1 DO
						IF receiveBuffer[idx]=0 THEN (*String delimiter found*)
							cbFrame:=idx+1;(*calculate length of received string*)
							MEMCPY(ADR(sFromClient), ADR(receiveBuffer),cbFrame); (*copy the received string to the output variable*)
							MEMMOVE(ADR(receiveBuffer), ADR(receiveBuffer[cbFrame]), cbReceived-cbFrame);(*move remaining data bytes*)
							dataReceived:=TRUE;  	(*Send an acknowledgement of data received*)
							state:=3; (*Move to the receive completion state*)
							endFound:=TRUE;
							EXIT;
						END_IF
					END_FOR
				ELSE(*no more free buffer space-overflow*)

					dataReceived:=FALSE;; (*Go to error state*)
					overflow:=TRUE;
					state:=4;
				END_IF
			ELSE(*no data received*)
					fbReceiveTON(IN:=FALSE, PT:=T#0ms);
					state:=1;
			END_IF
		ELSE(*error receiving data, exit function*)
			state:=4;
			dataReceived:=FALSE;
		END_IF
	END_IF

3:
	(*State used to process data*)
	velAxis1:=(STRING_TO_LREAL(MID(sFromClient, 7, 1)))/1000;  (*Extract the x distance*)
	velAxis2:=(STRING_TO_LREAL(MID(sFromClient, 7, 8)))/1000;
	velAxis3:=(STRING_TO_LREAL(MID(sFromClient, 7, 15)))/1000;
	velAxis4:=(STRING_TO_LREAL(MID(sFromClient, 7, 22)))/1000;

	fb_receive(bExecute:=FALSE); (*Reset the receive function*)
	startPos:=0; (*reset buffer beginning pointer*)
	endPos:=0;  (*reset buffer end pointer*)
	cbReceived:=0; (*reset bytes received counter*)
	sFromClient:=''; (*reset transition variable*)


	state:=1;
	RETURN;

4: (*Unused except for as an error state*)
trigger1:=FALSE;trigger2:=TRUE;

trigger2:=FALSE;

	(*Clear buffer-PROBABLY UNNECESSARY*)

	receiveBuffer[0]:=0;
	receiveBuffer[1]:=0;
	receiveBuffer[2]:=0;
	receiveBuffer[3]:=0;
	receiveBuffer[4]:=0;
	receiveBuffer[5]:=0;
	receiveBuffer[6]:=0;
	receiveBuffer[7]:=0;
	receiveBuffer[8]:=0;
	receiveBuffer[9]:=0;
	receiveBuffer[10]:=0;
	receiveBuffer[11]:=0;
	receiveBuffer[12]:=0;
	receiveBuffer[13]:=0;
	receiveBuffer[14]:=0;
	receiveBuffer[15]:=0;
	receiveBuffer[16]:=0;
	receiveBuffer[17]:=0;
	receiveBuffer[18]:=0;
	receiveBuffer[19]:=0;
	receiveBuffer[20]:=0;
	receiveBuffer[21]:=0;
	receiveBuffer[22]:=0;
	receiveBuffer[23]:=0;
	receiveBuffer[24]:=0;
	receiveBuffer[25]:=0;
	receiveBuffer[26]:=0;
	receiveBuffer[27]:=0;

	state:=1;
END_CASE;
END_FUNCTION_BLOCK

(* POU ROS_sendData, ST *)
FUNCTION_BLOCK ROS_sendData
VAR_INPUT
	sendBuffer: STRING;
	socketToUse: T_HSOCKET;
END_VAR
VAR_OUTPUT
END_VAR
VAR
 	(*Functions*)
	fb_send1: FB_SocketSend;
	(*Send data and variables*)
	sendBufferAddress1: DWORD;
	sendError1: UDINT;
END_VAR
(*
##
## This code was built by Christian Scheifele, University of Stuttgart, 2014.
## It  is derived in part from the TCP/IP server example on www.beckhoff.com
##
*)
	(*Send a greeting to the client*)
	sendBufferAddress1:=ADR(sendBuffer);
	(*Send information*)
	fb_send1
	(
		sSrvNetId:='',
		hSocket:=socketToUse,
		cbLen:=INT_TO_UDINT(LEN( sendBuffer ))+1,
		pSrc:=sendBufferAddress1,
		bExecute:=TRUE,
		tTimeout:=T#5s,
		nErrId=>sendError1,
	);

	fb_send1( bExecute := FALSE );
	fb_send1( bExecute := TRUE );
	fb_send1( bExecute := FALSE );
END_FUNCTION_BLOCK

(* POU ROS_convertSendData, ST *)
FUNCTION_BLOCK ROS_convertSendData
VAR_INPUT
	robotPosX: LREAL;
	robotPosY: LREAL;
	robotPosTheta: LREAL;
	robotVelX: LREAL;
	robotVelY: LREAL;
	robotVelTheta: LREAL;
END_VAR
VAR_OUTPUT
	send_message: STRING;
END_VAR
VAR
	posXString: STRING;
	posYString: STRING;
	posThetaString: STRING;
	velXString: STRING;
	velYString: STRING;
	velThetaString: STRING;
END_VAR
(*
##
## This code was built by Christian Scheifele, University of Stuttgart, 2014.
##
*)

(* Eingangsdaten verarbeiten *)
posXString := LREAL_TO_STRING(ABS(robotPosX));
posYString := LREAL_TO_STRING(ABS(robotPosY));
posThetaString := LREAL_TO_STRING(ABS(robotPosTheta)*100);
velXString := LREAL_TO_STRING(ABS(robotVelX));
velYString := LREAL_TO_STRING(ABS(robotVelY));
velThetaString := LREAL_TO_STRING(ABS(robotVelTheta)*100);

(* posXString bearbeiten *)
posXString := LEFT(posXString, FIND(posXString, '.')-1);
IF LEN(posXString) < 7 THEN
posXString := INSERT(posXString, '0000000',0 );
posXString := RIGHT(posXString, 6);
IF(robotPosX < 0) THEN
posXString := INSERT(posXString, '-',0 );
ELSE
posXString := INSERT(posXString, '0',0 );
END_IF;
END_IF;


(* posYString bearbeiten *)
posYString := LEFT(posYString, FIND(posYString, '.')-1);
IF LEN(posYString) < 7 THEN
	posYString := INSERT(posYString, '0000000',0 );
	posYString := RIGHT(posYString, 6);
	IF(robotPosY < 0) THEN
		posYString := INSERT(posYString, '-',0 );
	ELSE
		posYString := INSERT(posYString, '0',0 );
	END_IF;
END_IF;

(* posThetaString bearbeiten *)
posThetaString := LEFT(posThetaString, FIND(posThetaString, '.')-1);
IF LEN(posThetaString) < 7 THEN
	posThetaString := INSERT(posThetaString, '0000000',0 );
	posThetaString := RIGHT(posThetaString, 6);
	IF(robotPosTheta < 0) THEN
		posThetaString := INSERT(posThetaString, '-',0 );
	ELSE
		posThetaString := INSERT(posThetaString, '0',0 );
	END_IF;
END_IF;

(* velXString bearbeiten *)
velXString := LEFT(velXString, FIND(velXString, '.')-1);
IF LEN(velXString) < 7 THEN
velXString := INSERT(velXString, '0000000',0 );
velXString := RIGHT(velXString, 6);
	IF(robotVelX < 0) THEN
		velXString := INSERT(velXString, '-',0 );
	ELSE
		velXString := INSERT(velXString, '0',0 );
	END_IF;
END_IF;

(* velYString bearbeiten *)
velYString := LEFT(velYString, FIND(velYString, '.')-1);
IF LEN(velYString) < 7 THEN
velYString := INSERT(velYString, '0000000',0 );
velYString := RIGHT(velYString, 6);
	IF(robotVelY < 0) THEN
		velYString := INSERT(velYString, '-',0 );
	ELSE
		velYString := INSERT(velYString, '0',0 );
	END_IF;
END_IF;

(* velThetaString bearbeiten *)
velThetaString := LEFT(velThetaString, FIND(velThetaString, '.')-1);
IF LEN(velThetaString) < 7 THEN
velThetaString := INSERT(velThetaString, '0000000',0 );
velThetaString := RIGHT(velThetaString, 6);
	IF(robotVelTheta < 0) THEN
		velThetaString := INSERT(velThetaString, '-',0 );
	ELSE
		velThetaString := INSERT(velThetaString, '0',0 );
	END_IF;
END_IF;

send_message := CONCAT (posXString, posYString);
send_message := CONCAT (send_message, posThetaString);
send_message := CONCAT (send_message, velXString);
send_message := CONCAT (send_message, velYString);
send_message := CONCAT (send_message, velThetaString);
END_FUNCTION_BLOCK

(* POU jsConnect, ST *)
FUNCTION_BLOCK jsConnect
VAR


	(*Functions*)
	openSocket: BOOL:=FALSE;
	fb_listen: FB_SocketListen;
	fb_accept: FB_SocketAccept;
	(*Timers*)
	fbAcceptTON: TON;

	(*TCP socket variables*)
	activeSocketHandle: T_HSOCKET;
	socketHandle: T_HSOCKET;



	(*Error variables*)
	listenError: UDINT:=0;
	acceptError: UDINT;
	listenErrSet: BOOL;
	closeError: UDINT;
	sendError: UDINT;
	receiveError: UDINT;
	bSendError: BOOL;


	(*Trigger Variables*)
	bCloseAll: BOOL := TRUE;

	(*Connection information*)
	portNumber: INT:=8880;
	bAccepted: BOOL;

	(*Constants*)
	PLCPRJ_ACCEPT_POLLING_TIME: TIME:=T#1s;

	display: LREAL;
	heading: LREAL;

	state: INT:=0;

	xDist: LREAL;
	yDist: LREAL;
	zDist: LREAL;


	listening: BOOL;
	count: INT;
	fbresetTON: TON;
	timerOn: BOOL;
	timeUp: BOOL;
END_VAR
VAR_OUTPUT
	arduinoConnected: BOOL;
	socketToUse: T_HSOCKET;
END_VAR
trigger1:=FALSE; trigger2:=FALSE;
CASE state OF
0:

IF(fb_Listen.hListener.localAddr.nPort=portNumber) THEN
RETURN;

ELSE
state:=1;
END_IF

1:
(*This code was built by Chris Jarrett, Auckland University, 2014. It is derived in part from the TCP/IP server example on www.beckhoff.com*)
(*Listening State*)
(*Open a connection*)
(*Create socket and check for errors*)

fb_listen
(
	sSrvNetId:='' ,
	sLocalHost:='',
	nLocalPort:=portNumber,
	bExecute:=TRUE,
	tTimeout:=T#5s,
	hListener=>socketHandle,
	nErrId=>listenError,
	bError=>listenErrSet,

);

	IF(fb_Listen.hListener.localAddr.nPort=portNumber) THEN
		fb_listen(bExecute:=FALSE); 		(*Start listening and move to the accept state*)

		state:=2;
	ELSE
		(*Return to the listening state*)
		state:=1;
	END_IF



2:

(*Start accepting a client connection*)
fbAcceptTON( IN := TRUE, PT := T#2s);  (*Start a timer to poll for the accepted connection*)
		IF fbAcceptTON.Q THEN
			fbAcceptTON( IN := FALSE );	(*Reset timer*)
			fb_accept(  bExecute := FALSE  ); (*Generate a rising edge to activate the accept function*)
			fb_accept(hListener := socketHandle, bExecute:= TRUE, hSocket=>activeSocketHandle );
			state:=3; (*Move to the state where the client is accepted*)

			fbAcceptTON( IN := FALSE);

		END_IF
3:
(*Complete accpeting the client connection*)
	fb_accept( bExecute := FALSE ); (*Reset the accept function to try connection again if necessary*)
	IF NOT fb_accept.bBusy THEN
		IF NOT fb_accept.bError THEN
			IF fb_accept.bAccepted THEN
				bAccepted := TRUE; (*If the client connection is accepted without error then move to the send state*)
				fb_accept(bExecute:=FALSE);
				socketToUse:=fb_accept.hSocket;

				state:=4;
			ELSE
				fb_listen(bExecute:=FALSE);
				fb_accept(bExecute:=FALSE);
				arduinoConnected:=FALSE; (*If the connection attempt was not successful, return the boolean as false*)
				fbAcceptTON( IN := FALSE);
				state:=2;

				END_IF
		END_IF
	END_IF
4:
arduinoConnected:=TRUE;
RETURN;

END_CASE;
END_FUNCTION_BLOCK

(* POU jsDisconnect, ST *)
FUNCTION_BLOCK jsDisconnect
VAR_INPUT
	bCloseAll: BOOL;
END_VAR
VAR_OUTPUT
	connectionClosed: BOOL;
END_VAR
VAR
	fb_closeAll: FB_SocketCloseAll;
END_VAR
(*This function closes the TCP/IP port being used the Arduino connection*)

IF bCloseAll THEN
	bCloseAll:=FALSE;
	(*Close all open ports*)
	fb_closeAll(sSrvNetId:='', bExecute:=TRUE, tTimeOut:=T#5s );
ELSE
	fb_closeAll(bExecute:=FALSE);
END_IF


(*Move to the listening state*)
IF NOT fb_closeAll.bError THEN
	connectionClosed:=TRUE;


ELSE
connectionClosed:=FALSE;
END_IF
RETURN;
END_FUNCTION_BLOCK

(* POU jsReceiveData, ST *)
FUNCTION_BLOCK jsReceiveData
VAR_INPUT

	socketToUse: T_HSOCKET;
END_VAR
VAR_OUTPUT
	dataReceived: BOOL;
	botton: LREAL;
	xAxis: LREAL;
	yAxis: LREAL;
	zAxis: LREAL;
END_VAR
VAR
	(*Connection timers*)
	fbReceiveTON: TON;

 	(*Functions*)
	fb_receive: FB_SocketReceive;

	(*Send and receive data and variables*)
	receiveBuffer: ARRAY[0..19] OF BYTE;
	bytesReceived: UDINT;
	sendBuffer: STRING;
	sendBufferAddress: DWORD;
	cbReceived, startPos, endPos, idx : UDINT;
	cbFrame: UDINT;
	sFromClient: T_MaxString;
	overflow: BOOL;
	endFound: BOOL;

	(*Error variables*)
	acceptError: UDINT;
	receiveError: UDINT;

	state: INT:=1;
	xAsisString: STRING;
	yAsixString: STRING;
	zAxisString: STRING;
	bottonString: STRING;
	timerOn: BOOL;
	timeUp: BOOL;
	fbresetTON: TON;
END_VAR
CASE state OF
1:
(*Receive information*)
	fbReceiveTON(  IN := FALSE, PT:=T#0s); (*Receive first request immediately*)
	fbReceiveTON(  IN := TRUE ); (*Start a timer to ensure complete transfer of information*)

		IF fbReceiveTON.Q THEN
			fbReceiveTON(  IN := FALSE);
			fb_receive(bExecute:=FALSE);  (*Generate a rising edge to start receiving data*)
			fb_receive
			(
				sSrvNetId:='',
				hSocket :=socketToUse,
				cbLen:=SIZEOF(receiveBuffer)-cbReceived,
				pDest:=ADR(receiveBuffer)+cbReceived,
				tTimeout:=T#5s,
				nRecBytes=>bytesReceived,
				nErrId=>receiveError,
				bExecute:=TRUE,
			);

	(*Move to the receive completion state*)
	state:=2;
	END_IF

2:
(*Continue receiving data*)
	fb_receive( bExecute := FALSE );
	IF NOT fb_receive.bBusy THEN
		IF NOT fb_receive.bError THEN (*If no error has occurred then start the actual receiving of data*)

			IF (fb_receive.nRecBytes>0) THEN (*Bytes have been received*)

				startPos:=cbReceived; (*index of first data byte*)
				endPos:=cbReceived+fb_receive.nRecBytes-1; (*index of last byte*)
				cbReceived:=cbReceived+fb_receive.nRecBytes; (*Calculating the number of received data bytes*)
				cbFrame:=0; (*Reset the frame length*)


				IF cbReceived<SIZEOF(sFromClient) THEN (*no overflow*)
					fbReceiveTON(IN:=FALSE, PT:=T#0S);

					(*Search for the string delimiter(separation character for different strings)*)
					FOR idx:=startPos TO endPos BY 1 DO
						IF receiveBuffer[idx]=0 THEN (*String delimiter found*)
							cbFrame:=idx+1;(*calculate length of received string*)
							MEMCPY(ADR(sFromClient), ADR(receiveBuffer),cbFrame); (*copy the received string to the output variable*)
							MEMMOVE(ADR(receiveBuffer), ADR(receiveBuffer[cbFrame]), cbReceived-cbFrame);(*move remaining data bytes*)
							dataReceived:=TRUE;  	(*Send an acknowledgement of data received*)
							state:=3; (*Move to the receive completion state*)
							endFound:=TRUE;
							EXIT;
						END_IF
					END_FOR
				ELSE(*no more free buffer space-overflow*)

					dataReceived:=FALSE; (*Go to error state*)
					overflow:=TRUE;
					state:=4;
				END_IF
			ELSE(*no data received*)
					fbReceiveTON(IN:=FALSE, PT:=T#0ms);
					state:=1;
			END_IF
		ELSE(*error receiving data, exit function*)
			state:=4;
			dataReceived:=FALSE;
		END_IF
	END_IF

3:
	(*State used to process data*)
	botton:=(STRING_TO_LREAL(MID(sFromClient, 4, 1)));  (*Extract the x distance*)
IF(botton = 48) THEN
	xAxis:=((STRING_TO_LREAL(MID(sFromClient, 5, 5))-32768)/80);
	yAxis:=((STRING_TO_LREAL(MID(sFromClient, 5,10))-32768)/-80);
	zAxis:=((STRING_TO_LREAL(MID(sFromClient, 5, 15))-32768)/-80);
END_IF
IF(botton = 32)THEN
	yAxis:=((STRING_TO_LREAL(MID(sFromClient, 5, 5)))*40);
	xAxis:=((STRING_TO_LREAL(MID(sFromClient, 5,10)))*40);
	zAxis:=((STRING_TO_LREAL(MID(sFromClient, 5, 15)))*40);
END_IF

	fb_receive(bExecute:=FALSE); (*Reset the receive function*)
	startPos:=0; (*reset buffer beginning pointer*)
	endPos:=0;  (*reset buffer end pointer*)
	cbReceived:=0; (*reset bytes received counter*)
	sFromClient:=''; (*reset transition variable*)


	state:=1;
	RETURN;

4: (*Unused except for as an error state*)
trigger1:=FALSE; trigger2:=TRUE;  timerOn:=TRUE;(* reset arduino*)
fbresetTON(IN:=timerOn, PT:=REAL_TO_TIME(100), Q=>timeUp, ET=>);

IF (timeUp=TRUE)  THEN
trigger2:=FALSE;
timerOn:=FALSE;
END_IF

	(*Clear buffer-PROBABLY UNNECESSARY*)

	receiveBuffer[0]:=0;
	receiveBuffer[1]:=0;
	receiveBuffer[2]:=0;
	receiveBuffer[3]:=0;
	receiveBuffer[4]:=0;
	receiveBuffer[5]:=0;
	receiveBuffer[6]:=0;
	receiveBuffer[7]:=0;
	receiveBuffer[8]:=0;
	receiveBuffer[9]:=0;
	receiveBuffer[10]:=0;
	receiveBuffer[11]:=0;
	receiveBuffer[12]:=0;
	receiveBuffer[13]:=0;
	receiveBuffer[14]:=0;
	receiveBuffer[15]:=0;
receiveBuffer[16]:=0;
receiveBuffer[17]:=0;
receiveBuffer[18]:=0;
receiveBuffer[19]:=0;


	state:=1;


END_CASE;
END_FUNCTION_BLOCK

(* POU WP_connect, ST *)
FUNCTION_BLOCK WP_connect
VAR


	(*Functions*)
	openSocket: BOOL:=FALSE;
	fb_listen: FB_SocketListen;
	fb_accept: FB_SocketAccept;
	(*Timers*)
	fbAcceptTON: TON;

	(*TCP socket variables*)
	activeSocketHandle: T_HSOCKET;
	socketHandle: T_HSOCKET;



	(*Error variables*)
	listenError: UDINT:=0;
	acceptError: UDINT;
	listenErrSet: BOOL;
	closeError: UDINT;
	sendError: UDINT;
	receiveError: UDINT;
	bSendError: BOOL;


	(*Trigger Variables*)
	bCloseAll: BOOL := TRUE;

	(*Connection information*)
	portNumber: INT:=8800;
	bAccepted: BOOL;

	(*Constants*)
	PLCPRJ_ACCEPT_POLLING_TIME: TIME:=T#1s;

	display: LREAL;
	heading: LREAL;

	state: INT:=0;

	xDist: LREAL;
	yDist: LREAL;
	zDist: LREAL;


	listening: BOOL;
	count: INT;
	fbresetTON: TON;
	timerOn: BOOL;
	timeUp: BOOL;
END_VAR
VAR_OUTPUT
	WPConnected: BOOL;
	socketToUse: T_HSOCKET;
END_VAR
trigger1:=FALSE; trigger2:=FALSE;
CASE state OF
0:

IF(fb_Listen.hListener.localAddr.nPort=portNumber) THEN
RETURN;

ELSE
state:=1;
END_IF

1:
(*This code was built by Chris Jarrett, Auckland University, 2014. It is derived in part from the TCP/IP server example on www.beckhoff.com*)
(*Listening State*)
(*Open a connection*)
(*Create socket and check for errors*)

fb_listen
(
	sSrvNetId:='' ,
	sLocalHost:='',
	nLocalPort:=portNumber,
	bExecute:=TRUE,
	tTimeout:=T#5s,
	hListener=>socketHandle,
	nErrId=>listenError,
	bError=>listenErrSet,

);

	IF(fb_Listen.hListener.localAddr.nPort=portNumber) THEN
		fb_listen(bExecute:=FALSE); 		(*Start listening and move to the accept state*)

		state:=2;
	ELSE
		(*Return to the listening state*)
		state:=1;
	END_IF



2:

(*Start accepting a client connection*)
fbAcceptTON( IN := TRUE, PT := T#2s);  (*Start a timer to poll for the accepted connection*)
		IF fbAcceptTON.Q THEN
			fbAcceptTON( IN := FALSE );	(*Reset timer*)
			fb_accept(  bExecute := FALSE  ); (*Generate a rising edge to activate the accept function*)
			fb_accept(hListener := socketHandle, bExecute:= TRUE, hSocket=>activeSocketHandle );
			state:=3; (*Move to the state where the client is accepted*)

			fbAcceptTON( IN := FALSE);

		END_IF
3:
(*Complete accpeting the client connection*)
	fb_accept( bExecute := FALSE ); (*Reset the accept function to try connection again if necessary*)
	IF NOT fb_accept.bBusy THEN
		IF NOT fb_accept.bError THEN
			IF fb_accept.bAccepted THEN
				bAccepted := TRUE; (*If the client connection is accepted without error then move to the send state*)
				fb_accept(bExecute:=FALSE);
				socketToUse:=fb_accept.hSocket;

				state:=4;
			ELSE
				fb_listen(bExecute:=FALSE);
				fb_accept(bExecute:=FALSE);
				WPConnected:=FALSE; (*If the connection attempt was not successful, return the boolean as false*)
				fbAcceptTON( IN := FALSE);
				state:=2;

				END_IF
		END_IF
	END_IF
4:
WPConnected:=TRUE;
RETURN;

END_CASE;
END_FUNCTION_BLOCK

(* POU WP_Disconnect, ST *)
FUNCTION_BLOCK WP_Disconnect
VAR_INPUT
	bCloseAll: BOOL;
END_VAR
VAR_OUTPUT
	connectionClosed: BOOL;
END_VAR
VAR
	fb_closeAll: FB_SocketCloseAll;
END_VAR
(*This function closes the TCP/IP port being used the Arduino connection*)

IF bCloseAll THEN
	bCloseAll:=FALSE;
	(*Close all open ports*)
	fb_closeAll(sSrvNetId:='', bExecute:=TRUE, tTimeOut:=T#5s );
ELSE
	fb_closeAll(bExecute:=FALSE);
END_IF


(*Move to the listening state*)
IF NOT fb_closeAll.bError THEN
	connectionClosed:=TRUE;


ELSE
connectionClosed:=FALSE;
END_IF
RETURN;
END_FUNCTION_BLOCK

(* POU WP_ReceiveData, ST *)
FUNCTION_BLOCK WP_ReceiveData
VAR_INPUT

	socketToUse: T_HSOCKET;
END_VAR
VAR_OUTPUT
	dataReceived: BOOL;
	botton: INT;
	xAxis: LREAL;
	yAxis: LREAL;
	zAxis: LREAL;
END_VAR
VAR
	(*Connection timers*)
	fbReceiveTON: TON;

 	(*Functions*)
	fb_receive: FB_SocketReceive;

	(*Send and receive data and variables*)
	receiveBuffer: ARRAY[0..0] OF BYTE;
	bytesReceived: UDINT;
	sendBuffer: STRING;
	sendBufferAddress: DWORD;
	cbReceived, startPos, endPos, idx : UDINT;
	cbFrame: UDINT;
	sFromClient: T_MaxString;
	overflow: BOOL;
	endFound: BOOL;

	(*Error variables*)
	acceptError: UDINT;
	receiveError: UDINT;

	state: INT:=1;
	xAxisString: STRING;
	yAxixString: STRING;
	zAxisString: STRING;
	bottonString: STRING;
	timerOn: BOOL;
	timeUp: BOOL;
	fbresetTON: TON;
END_VAR
CASE state OF
1:
(*Receive information*)
	fbReceiveTON(  IN := FALSE, PT:=T#0s); (*Receive first request immediately*)
	fbReceiveTON(  IN := TRUE ); (*Start a timer to ensure complete transfer of information*)

		IF fbReceiveTON.Q THEN
			fbReceiveTON(  IN := FALSE);
			fb_receive(bExecute:=FALSE);  (*Generate a rising edge to start receiving data*)
			fb_receive
			(
				sSrvNetId:='',
				hSocket :=socketToUse,
				cbLen:=SIZEOF(receiveBuffer)-cbReceived,
				pDest:=ADR(receiveBuffer)+cbReceived,
				tTimeout:=T#5s,
				nRecBytes=>bytesReceived,
				nErrId=>receiveError,
				bExecute:=TRUE,
			);

	(*Move to the receive completion state*)
	state:=2;
	END_IF

2:
(*Continue receiving data*)
	fb_receive( bExecute := FALSE );
	IF NOT fb_receive.bBusy THEN
		IF NOT fb_receive.bError THEN (*If no error has occurred then start the actual receiving of data*)

			IF (fb_receive.nRecBytes>0) THEN (*Bytes have been received*)

				startPos:=cbReceived; (*index of first data byte*)
				endPos:=cbReceived+fb_receive.nRecBytes-1; (*index of last byte*)
				cbReceived:=cbReceived+fb_receive.nRecBytes; (*Calculating the number of received data bytes*)
				cbFrame:=0; (*Reset the frame length*)


				IF cbReceived<SIZEOF(sFromClient) THEN (*no overflow*)
					fbReceiveTON(IN:=FALSE, PT:=T#0S);

					(*Search for the string delimiter(separation character for different strings)*)
					FOR idx:=startPos TO endPos BY 1 DO
						IF receiveBuffer[idx]=0 THEN (*String delimiter found*)
							cbFrame:=idx+1;(*calculate length of received string*)
							MEMCPY(ADR(sFromClient), ADR(receiveBuffer),cbFrame); (*copy the received string to the output variable*)
							MEMMOVE(ADR(receiveBuffer), ADR(receiveBuffer[cbFrame]), cbReceived-cbFrame);(*move remaining data bytes*)
							dataReceived:=TRUE;  	(*Send an acknowledgement of data received*)
							state:=3; (*Move to the receive completion state*)
							endFound:=TRUE;
							EXIT;
						END_IF
					END_FOR
				ELSE(*no more free buffer space-overflow*)

					dataReceived:=FALSE; (*Go to error state*)
					overflow:=TRUE;
					state:=4;
				END_IF
			ELSE(*no data received*)
					fbReceiveTON(IN:=FALSE, PT:=T#0ms);
					state:=1;
			END_IF
		ELSE(*error receiving data, exit function*)
			state:=4;
			dataReceived:=FALSE;
		END_IF
	END_IF

3:
	(*State used to process data*)	(*State used to process data*)
	botton:=(STRING_TO_INT(MID(sFromClient, 1, 1)));  (*Extract the x distance*)

	CASE botton OF
		1:
			xAxis := 0;
			yAxis := 0;
			zAxis := 600;
		2:
			xAxis := 0;
			yAxis := 600;
			zAxis := 0;
		3:
			xAxis := 0;
			yAxis := 0;
			zAxis := -600;
		4:
			xAxis := -600;
			yAxis := 0;
			zAxis := 0;
		5:
			xAxis := 0;
			yAxis := 0;
			zAxis := 0;
		6:
			xAxis := 600;
			yAxis := 0;
			zAxis := 0;
		8:
			xAxis := 0;
			yAxis := -600;
			zAxis := 0;
		ELSE
			xAxis:= 0;
			yAxis:= 0;
			zAxis:= 0;
		END_CASE

	fb_receive(bExecute:=FALSE); (*Reset the receive function*)
	startPos:=0; (*reset buffer beginning pointer*)
	endPos:=0;  (*reset buffer end pointer*)
	cbReceived:=0; (*reset bytes received counter*)
	sFromClient:=''; (*reset transition variable*)


	state:=1;
	RETURN;

4: (*Unused except for as an error state*)
trigger1:=FALSE; trigger2:=TRUE;  timerOn:=TRUE;(* reset arduino*)
fbresetTON(IN:=timerOn, PT:=REAL_TO_TIME(100), Q=>timeUp, ET=>);

IF (timeUp=TRUE)  THEN
trigger2:=FALSE;
timerOn:=FALSE;
END_IF

	(*Clear buffer-PROBABLY UNNECESSARY*)

	receiveBuffer[0]:=0;
	state:=1;


END_CASE;
END_FUNCTION_BLOCK

(* POU MainFast, ST *)
PROGRAM MainFast
VAR
	fblocalization:  localization;
END_VAR
fblocalization(robotPosX=>robotPosX, robotPosY=>robotPosY,robotPosTheta=>robotPosTheta, robotVelX=>robotVelX, robotVelY=>robotVelY, robotVelTheta=>robotVelTheta);
END_PROGRAM

(* POU localization, ST *)
FUNCTION_BLOCK localization  (* to be call by fb movement only*)  (* calls  fb kalman filter*)
VAR_INPUT
END_VAR
VAR_OUTPUT
(*for ROS*)
	robotPosX:	LREAL;
	robotPosY:	LREAL;
	robotPosTheta:	LREAL;
	robotVelX:	LREAL;
	robotVelY:	LREAL;
	robotVelTheta:	LREAL;
END_VAR
VAR
(* from wheel motor encoder*)
	w1:LREAL;
	w2:LREAL;
	w3:LREAL;
	w4:LREAL;
	sw1: LREAL;
	sw2: LREAL;
	sw3: LREAL
;	sw4: LREAL;

	encoder1: AXIS_REF;
	encoder2: AXIS_REF;
	encoder3: AXIS_REF;
	encoder4: AXIS_REF;

(*working variable*)
	globalePosX:	LREAL;
	globalePosY:	LREAL;heading_radians1: LREAL;
	globalePosX1:	LREAL;
	globalePosY1:	LREAL;
	sencoderX:	ARRAY[1..5] OF		LREAL;
	sencoderY:	ARRAY[1..5] OF		LREAL;
	sheading:	ARRAY[1..5] OF		LREAL;
(*kalman filter*)
	fbkalmanFilter:	ARRAY[1..3] OF 	kalmanFilter;
	fbekalmanFilter:	ARRAY[1..3] OF 	extendedKalmanFilter;
	fbTON3:	TON;
	startTimer3: BOOL;
	timer3On: BOOL;
(*heading*)
	A:LREAL;
	q: INT;
	differentX: LREAL;
	differentY: LREAL;

(*Arduino variables*)
	arduinoCalculate1:				arduinoCalculation;
	xDistA: LREAL;
	yDistA: LREAL;
	headingA: LREAL;

(*velocity calculation*)
	combinedXOld: LREAL:=0;
	combinedYOld: LREAL:=0;
	combinedHOld: LREAL:=0;
	count:INT;
	velocityX: LREAL;
	velocityY: LREAL;
	velocityH: LREAL;

END_VAR
(* from wheel motor encoder*)
w1:=axis1.NcToPlc.ActPos;
w2:=-axis2.NcToPlc.ActPos;
w3:=axis3.NcToPlc.ActPos;
w4:=-axis4.NcToPlc.ActPos;
encoderY[5]:=0.025*((w1-sw1)+(w2-sw2)+(w3-sw3)+(w4-sw4))*1.634*1.006;
encoderX[5]:=-0.025*((w1-sw1)-(w2-sw2)-(w3-sw3)+(w4-sw4))*1.339*1.006;
heading[5]:=(-0.025*(-(w1-sw1)+(w2-sw2)-(w3-sw3)+(w4-sw4))*0.144)+90;


(* set ALL to zero at start of motion*)
IF (home) THEN
sencoderX[3]:=0.0;
sencoderX[1]:=encoder1.NcToPlc.ActPos;
sencoderX[2]:=encoder3.NcToPlc.ActPos;
xDistA:=0;
yDistA:=0;
sencoderX[4]:=0;
encoderX[4]:=0;
sencoderY[3]:=0.0;
sencoderY[1]:=encoder2.NcToPlc.ActPos;
sencoderY[2]:=encoder4.NcToPlc.ActPos;
sencoderY[4]:=0;
encoderY[4]:=0;
heading[1]:=0.0;
sheading[4]:=headingA;
sw1:=axis1.NcToPlc.ActPos;
sw2:=-axis2.NcToPlc.ActPos;
sw3:=axis3.NcToPlc.ActPos;
sw4:=-axis4.NcToPlc.ActPos;
globalePosX:=0;
globalePosY:=0;
home:=FALSE;
END_IF

(* continue to read data*)
	encoderX[1]:=(encoder1.NcToPlc.ActPos - sencoderX[1]);
	encoderY[1]:=(encoder2.NcToPlc.ActPos - sencoderY[1]);

	encoderX[2]:=(encoder3.NcToPlc.ActPos - sencoderX[2]);
	encoderY[2]:=(encoder4.NcToPlc.ActPos - sencoderY[2]);


(*Heading1 calculation from encoder 2 and 3, assume encoder 2 at origin*)
	differentX:=encoderX[2]-encoderX[1]-0.2;
	differentY:=encoderY[2]-encoderY[1]+550;

	IF (differentX>=0 AND differentY>=0) THEN A:=ATAN(differentY/differentX)*180/3.142; heading[1]:=180-(A-(0.03)); Q:=1; 		(* 1st quad*)
	ELSIF (differentX<0 AND differentY>=0) THEN A:=ATAN(differentY/-differentX)*180/3.142;heading[1]:=180-(180-A-(0.03)); Q:=2;  (* 2nd quad*)
	ELSIF (differentX<0 AND differentY<0) THEN A:=ATAN(differentY/differentX)*180/3.142; heading[1]:=180-(180+A-(0.03));    Q:=3;	(* 3rd quad*)
	ELSIF (differentX>=0 AND differentY<0) THEN A:=ATAN(-differentY/differentX)*180/3.142; heading[1]:=180-(360-A-(0.03)); Q:=4;   	(* 4th quad*)
	END_IF
IF heading[1] < -180 THEN heading[1]:=heading[1]+360; END_IF
IF heading[1] > 180 THEN heading[1]:=heading[1]-360;   END_IF(* heading is always between +180 to -180*)



(*kalman filter.   cycle time = 10 ms*)
(*IF (trigger1=TRUE AND timer3On=FALSE) THEN*)
fbTON3(IN:=startTimer3, PT:=LREAL_TO_TIME(10) , Q=>timer3On);
count:=count+1;
IF (count>0) THEN startTimer3:=TRUE; END_IF
	IF (timer3On=TRUE) THEN
	timer3On:=FALSE;
	startTimer3:=FALSE;
	count:=0;
(* kalman filter to combine the spherical ball encoder [1] to the wheel encoder[5] combined signal =[3]*)
	fbkalmanFilter[1](reading:=(encoderX[1]-encoderX[5]),target:=0,noiseVar:= 0.1);    (* encoder in mm noise var need to vadify*)
	encoderX[3]:=fbkalmanFilter[1].out+encoderX[5];
	fbkalmanFilter[2](reading:=(encoderY[1]-encoderY[5]),target:=0,noiseVar:= 0.1);
	encoderY[3]:=fbkalmanFilter[2].out+encoderY[5];
	fbkalmanFilter[3](reading:=(heading[1]-heading[5]),target:=0,noiseVar:= 0.1);
	heading[3]:=fbkalmanFilter[3].out+heading[5];
(*convert to world*)
	heading_radians1 :=  heading[3]/180 * 3.1415963;
	globalePosX1 := globalePosX1 + SIN(heading_radians1) *( encoderX[3] -combinedXOld) +  COS(heading_radians1) * (encoderY[3] - combinedYOld);
	globalePosY1 := globalePosY1 + SIN(heading_radians1) * (encoderY[3] - combinedYOld) - COS(heading_radians1) *( encoderX[3] -combinedXOld);

	combinedXOld:=encoderX[3];
	combinedYOld:=encoderY[3];
(* arduino*)
	arduinoCalculate1(xDistA=>xDistA, yDistA=>ydistA,	headingA=>headingA);
	encoderX[4]:=xDistA+sencoderX[4];
	encoderY[4]:=yDistA +sencoderY[4];
	heading[4]:=headingA-sheading[4]+90;
	IF (trigger1 = FALSE) THEN sencoderX[4]:=encoderX[4]; sencoderY[4]:=encoderY[4];END_IF

	fbekalmanFilter[1](reading:=(encoderX[4]-globalePosX1),target:=0,noiseVar:= 0.1);
	globalePosX:=fbekalmanFilter[1].out+globalePosX1;
	fbekalmanFilter[2](reading:=(encoderY[4]-globalePosY1),target:=0,noiseVar:= 0.1);
	globalePosY:=fbekalmanFilter[2].out+globalePosY1;
	fbekalmanFilter[3](reading:=(heading[4]-heading[3]),target:=0,noiseVar:= 0.1);
	combinedH:=fbekalmanFilter[3].out+heading[3];

	velocityX:=(combinedX-combinedXOld)/0.01;
	velocityY:=(combinedY-combinedYOld)/0.01;
	velocityH:=(combinedH-combinedHOld)/0.01;



	END_IF


(*output*)
robotPosTheta:=combinedH;
robotPosX:=globalePosX;
robotPosY:=globalePosY;
robotVelX:=velocityX;
robotVelY:=velocityY;
robotVelTheta:=velocityH;


(* combining encoders  *)
(* set ALL to zero at start of motion
IF motorRunning=TRUE  THEN start:=TRUE; END_IF
IF motorRunning = FALSE THEN start:=FALSE;  END_IF
fbR_trig(clk:=start,Q=>startMotion);
fbF_trig(clk:=start,Q=>stopMotion);
IF (startMotion=TRUE)    (*capture the starting value*)
THEN
exPosition:=directionToMove;
sencoderX[1]:=0.0;
sencoderX[2]:=axis[5].NcToPlc.ActPos;
sencoderX[3]:=axis[7].NcToPlc.ActPos;
sencoderY[1]:=0.0;
sencoderY[2]:=axis[6].NcToPlc.ActPos;
sencoderY[3]:=axis[8].NcToPlc.ActPos;

startMotion:=FALSE;                  (* so that this initialization only do once*)
END_IF

(* ignore all the data from direction that do not move*)

	encoderX[2]:=(axis[5].NcToPlc.ActPos - sencoderX[2]);
	encoderX[3]:=(axis[7].NcToPlc.ActPos - sencoderX[3]);

	encoderY[2]:=(axis[6].NcToPlc.ActPos - sencoderY[2]);
	encoderY[3]:=(axis[8].NcToPlc.ActPos - sencoderY[3]);

(*Kalman Filter: startKF do a loop every 10ms, updating the position (encoder 1 and 2 and 3) every 10ms*)

IF (motorRunning=TRUE)   THEN
	startKF:=TRUE;
	startTimer2:=TRUE;   (*timer 2 is for calculating encoder 1*)
ELSE
	startKF:=FALSE;
	startTimer2:=FALSE;
END_IF

(* use motor motion as ref = encoder [1] *)

fbTON2(IN:=startTimer2, PT:=timeToMove , ET=>ET2);

	CASE exPosition OF
	1: encoderX[1]:=distanceToMove*-1000*(4.0/6.4)*TIME_TO_LREAL(ET2)/TIME_TO_LREAL(timeToMove);encoderY[1]:=distanceToMove*1000*(5.0/6.4)*TIME_TO_LREAL(ET2)/ TIME_TO_LREAL(timeToMove);
	2: encoderX[1]:=0.0; encoderY[1]:=distanceTomove*1000*TIME_TO_LREAL(ET2)/ TIME_TO_LREAL(timeToMove);
	3: encoderX[1]:=distanceToMove*1000*(4.0/6.4)*TIME_TO_LREAL(ET2)/TIME_TO_LREAL (timeToMove); encoderY[1]:=distanceToMove*1000*(5.0/6.4)*TIME_TO_LREAL(ET2)/ TIME_TO_LREAL(timeToMove);
	4: encoderX[1]:=distanceToMove*-1000*TIME_TO_LREAL(ET2)/TIME_TO_LREAL (timeToMove); encoderY[1]:=0;
	5: encoderX[1]:=distanceToMove*1000*TIME_TO_LREAL(ET2)/TIME_TO_LREAL (timeToMove); encoderY[1]:=0;
	6: encoderX[1]:=distanceToMove*-1000*(4.0/6.4)*TIME_TO_LREAL(ET2)/TIME_TO_LREAL (timeToMove); encoderY[1]:=distanceToMove*-1000*(5.0/6.4)*TIME_TO_LREAL(ET2)/ TIME_TO_LREAL(timeToMove);
	7: encoderX[1]:=0.0; encoderY[1]:=distanceTomove*-1000*TIME_TO_LREAL(ET2)/TIME_TO_LREAL (timeToMove);
	8:encoderX[1]:=distanceToMove*1000*(4.0/6.)*TIME_TO_LREAL(ET2)/TIME_TO_LREAL (timeToMove); encoderY[1]:=distanceToMove*1000*(5.0/6.4)*TIME_TO_LREAL(ET2)/TIME_TO_LREAL (timeToMove);
	9:encoderX[1]:=0.0; encoderY[1]:=0.0;
	10:encoderX[1]:=0.0; encoderY[1]:=0.0;
	ELSE
	encoderX[1]:=0.0; encoderY[1]:=0.0;
	END_CASE
encoderX[4]:=(inertialxDist*TIME_TO_LREAL(ET2)+20)/1000;
encoderY[4]:=(inertialyDist*TIME_TO_LREAL(ET2)+20)/1000;
IF(startKF=TRUE AND timer3On=FALSE) THEN startTimer3:= TRUE; ELSE startTimer3:=FALSE; END_IF

fbTON3(IN:=startTimer3, PT:=LREAL_TO_TIME(10) , Q=>timer3On);
	IF (timer3On=TRUE) THEN
	fbkalmanFilter[1](reading:=(encoderX[3]),target:=encoderX[1],noiseVar:= 0.1);    (* encoder in mm*)
	combinedX:=fbkalmanFilter[1].out;
	fbkalmanFilter[2](reading:=(encoderY[3]),target:=encoderY[1],noiseVar:= 0.1);
	combinedY:=fbkalmanFilter[2].out;
	startTimer3:=FALSE;
	END_IF

IF (stopMotion=TRUE) THEN

	(*encoderX[4]:=inertialxDist-sencoderX[4];
	encoderY[4]:=inertialyDist-sencoderY[4];*)
	heading[2]:= inertialheading;

	stopMotion:=FALSE;   (*do only once*)


(*average*)
IF(main.startLoop=TRUE) THEN oldCombinedX:=combinedX; oldCombinedY:=combinedY; oldCombinedH:=combinedH; ELSE oldCombinedX:=0; oldCombinedY:=0; END_IF

	combinedX:=oldCombinedX+(combinedX*1.0+encoderX[4]*0.00);
	combinedY:=oldCombinedY+(combinedY*1.0+encoderY[4]*0.00);
	IF (heading[1]-heading[2]<300 AND heading[1]-heading[2]>-300)
	THEN combinedH:=oldCombinedH+((heading[1]+heading[2]) / 2);
	ELSE
	combinedH:=oldCombinedH+(heading[1]+heading[2]);  (*cater for the angle such as 350 and 10*)
		IF combinedH>=360.0 THEN combinedH:=combinedH-360; END_IF
	END_IF
END_IF

(*Heading1 calculation from encoder 2 and 3, assume encodr 2 at origin*)
	differentX:=encoderX[3]-encoderX[2]+70;
	differentY:=520+encoderY[3]-encoderY[2];

	IF (differentX>=0 AND differentY>=0) THEN heading[1]:=90-(ATAN(differentY/differentX))*3.142/180+7.67;  		(* 1st quad*)
	ELSIF (differentX<0 AND differentY>=0) THEN heading[1]:=270-(ATAN(differentY/differentX))*3.142/180+7.67;   	(* 2nd quad*)
	ELSIF (differentX<0 AND differentY<0) THEN heading[1]:=270-(ATAN(differentY/differentX))*3.142/180+7.67;     	(* 3rd quad*)
	ELSIF (differentX>=0 AND differentY<0) THEN heading[1]:=90+(ATAN(differentY/differentX))*3.142/180+7.67;    	(* 4th quad*)
	END_IF*)
RETURN;
END_FUNCTION_BLOCK

(* POU kalmanFilter, ST *)
FUNCTION_BLOCK kalmanFilter
VAR_INPUT
	reading: LREAL;
	target: LREAL;
	noiseVar: LREAL;
END_VAR
VAR_OUTPUT
	out: LREAL;
END_VAR
VAR
	control: LREAL;
	oldP: LREAL;
	newP: LREAL := 1.0;
	oldX: LREAL;
	newX: LREAL:=0.0;
	K: LREAL;
	oldPredict: LREAL:=0.0;

END_VAR
control:=target-NewX;
(* timeupdate*)

oldP :=newP;
oldX:=newX+control;

(*measurement update*)

K:=oldP / (oldP+noiseVar);
NewX:=oldX+K*(reading-oldX);
newP:=(1-K)*oldP;
out:=NewX;

RETURN;
END_FUNCTION_BLOCK

(* POU extendedKalmanFilter, ST *)
FUNCTION_BLOCK extendedKalmanFilter
VAR_INPUT
	reading: LREAL;
	target: LREAL;
	noiseVar: LREAL;
END_VAR
VAR_OUTPUT
	out: LREAL;
END_VAR
VAR
	control: LREAL;
	estP: LREAL;
	newP: LREAL := 1.0;
	estX: LREAL;
	newX: LREAL:=0.0;
	newK: LREAL;
	oldPredict: LREAL:=0.0;
	count:INT;

(*extened KF*)
	F: LREAL:=1.0;
	H: LREAL:=1.0;
	oldfuncH: LREAL;
	funcH:LREAL;
	oldfuncF: LREAL;
	funcF: LREAL;
	oldX: LREAL;
	oldestX: LREAL;
END_VAR
(*kalman filter.   cycle time = 10 ms;   added f and h for extended KF assume B = 1*)
control:=target-NewX;
count:=count+1;

(* timeupdate*)
oldfuncF:=funcF;
funcF:=F*newX;
IF (newX-oldX<>0) THEN F:=(funcF-oldfuncF)/(newX-oldX); END_IF
estP :=F*newP*F;  (* assume Q =0 *)
oldestX:=estX;
estX:=funcF+control;

(*measurement update*)
newK:=H*estP / (H*estP*H+noiseVar);

oldfuncH:=funcH;
funcH:=H*estX;
IF (estX-oldestX<>0) THEN H:=(funcH-oldfuncH)/(estX-oldestX); END_IF
oldX:=newX;
newX:=estX+newK*(reading-funcH);
newP:=(1-newK*H)*estP;
out:=NewX;

RETURN;
END_FUNCTION_BLOCK

(* POU arduinoCalculation, ST *)
FUNCTION_BLOCK arduinoCalculation
VAR_INPUT

END_VAR
VAR_OUTPUT
	xDistA: LREAL;
	yDistA: LREAL;
	headingA: LREAL;
END_VAR
VAR
	connectArduino1:				ArduinoConnect;
	disconnectArduino1:			ArduinoDisconnect;
	receiveData1:				ArduinoReceiveData;

	tcpSocket: T_HSOCKET;
	connectionOpen: BOOL:=FALSE;
	closeConnection: BOOL:=TRUE;
	dataReceived: BOOL;
	heading: LREAL;
	xAccA: ARRAY[1..10] OF LREAL;
	yAccA: ARRAY[1..10] OF LREAL;
	xBias: LREAL;
	yBias: LREAL;
	xAccel: LREAL;
	yAccel: LREAL;
	xVel:LREAL;
	yVel:LREAL;
	xPVel: LREAL:=0;
	yPVel:LREAL:=0;
	xPDist: LREAL;
	yPDist:LREAL;
	j: INT:=0;
	aMove:BOOL;
END_VAR
(*Arduino*)
(*Close TCP port from last time-remove after DEBUG*)
IF closeConnection THEN
	disconnectArduino1(bCloseAll:=closeConnection);
	closeConnection:=FALSE;
END_IF

(*Open a connection*)
IF (connectionOpen=FALSE) THEN
	connectArduino1(arduinoConnected=>connectionOpen, socketToUse=>tcpSocket);
END_IF

IF (connectionOpen=TRUE) THEN
	receiveData1(socketToUse:=tcpSocket,dataReceived=>dataReceived,heading=>headingA, xAccel=>xAccel, yAccel=>yAccel);
END_IF
(* Calculation*)
IF (dataReceived) THEN

IF (trigger1=FALSE AND aMove = FALSE) THEN
xAccA[1]:= xAccel; yAccA[1]:=yAccel;
xAccA[2]:= xAccA[1]; yAccA[2]:=yAccA[1];
xAccA[3]:= xAccA[2]; yAccA[3]:=yAccA[2];
xAccA[4]:= xAccA[3]; yAccA[4]:=yAccA[3];
xAccA[5]:= xAccA[4]; yAccA[5]:=yAccA[4];
xAccA[6]:= xAccA[5]; yAccA[6]:=yAccA[5];
xAccA[7]:= xAccA[6]; yAccA[7]:=yAccA[6];
xAccA[8]:= xAccA[7]; yAccA[8]:=yAccA[7];
xAccA[9]:= xAccA[8]; yAccA[9]:=yAccA[8];
xAccA[10]:= xAccA[9]; yAccA[10]:=yAccA[9];
xBias:=(xAccA[1]+xAccA[2]+xAccA[3]+xAccA[4]+xAccA[5]+xAccA[6]+xAccA[7]+xAccA[8]+xAccA[9]+xAccA[10])/10;
yBias:=(yAccA[1]+yAccA[2]+yAccA[3]+yAccA[4]+yAccA[5]+yAccA[6]+yAccA[7]+yAccA[8]+yAccA[9]+yAccA[10])/10;
END_IF

	IF (trigger1 =TRUE) THEN
		IF (aMove=FALSE) THEN xDistA:=0; yDistA:=0; aMove:=TRUE;END_IF (*start*)

  		IF (trigger2=FALSE ) THEN
		xAccA[1]:= xAccel; yAccA[1]:=yAccel;
		xVel:=(xAccA[1]-xBias)/16384*9.81*0.01+xVel; yVel:=(yAccA[1]-yBias)/16384*9.81*0.01+yVel;
		xPVel := xVel; yPVel:=yVel;
		ELSE
		xVel:=xPVel; yVel:=yPVel;
		END_IF
	xDistA:=(xVel)*10+xDistA;  yDistA:=(yVel)*10+yDistA;
	ELSE
	xAccA[1]:=0; yACCA[1]:=0;
	xVel:=0; yVel:=0;
	yPVel:=0;xPVel:=0;
	END_IF

	IF (trigger1 =FALSE AND aMove=TRUE) THEN  (*stop*)
	aMove:=FALSE;
	END_IF
END_IF


RETURN;
END_FUNCTION_BLOCK

(* POU ArduinoConnect, ST *)
FUNCTION_BLOCK ArduinoConnect
VAR


	(*Functions*)
	openSocket: BOOL:=FALSE;
	fb_listen: FB_SocketListen;
	fb_accept: FB_SocketAccept;
	(*Timers*)
	fbAcceptTON: TON;

	(*TCP socket variables*)
	activeSocketHandle: T_HSOCKET;
	socketHandle: T_HSOCKET;



	(*Error variables*)
	listenError: UDINT:=0;
	acceptError: UDINT;
	listenErrSet: BOOL;
	closeError: UDINT;
	sendError: UDINT;
	receiveError: UDINT;
	bSendError: BOOL;


	(*Trigger Variables*)
	bCloseAll: BOOL := TRUE;

	(*Connection information*)
	portNumber: INT:=8888;
	bAccepted: BOOL;

	(*Constants*)
	PLCPRJ_ACCEPT_POLLING_TIME: TIME:=T#1s;

	display: LREAL;
	heading: LREAL;

	state: INT:=0;

	xDist: LREAL;
	yDist: LREAL;
	zDist: LREAL;


	listening: BOOL;
	count: INT;
	fbresetTON: TON;
	timerOn: BOOL;
	timeUp: BOOL;
END_VAR
VAR_OUTPUT
	arduinoConnected: BOOL;
	socketToUse: T_HSOCKET;
END_VAR
CASE state OF
0:

IF(fb_Listen.hListener.localAddr.nPort=portNumber) THEN
RETURN;

ELSE
state:=1;
END_IF

1:
(*This code was built by Chris Jarrett, Auckland University, 2014. It is derived in part from the TCP/IP server example on www.beckhoff.com*)
(*Listening State*)
(*Open a connection*)
(*Create socket and check for errors*)

fb_listen
(
	sSrvNetId:='' ,
	sLocalHost:='',
	nLocalPort:=portNumber,
	bExecute:=TRUE,
	tTimeout:=T#5s,
	hListener=>socketHandle,
	nErrId=>listenError,
	bError=>listenErrSet,

);

	IF(fb_Listen.hListener.localAddr.nPort=portNumber) THEN
		fb_listen(bExecute:=FALSE); 		(*Start listening and move to the accept state*)

		state:=2;
	ELSE
		(*Return to the listening state*)
		state:=1;
	END_IF



2:

(*Start accepting a client connection*)
fbAcceptTON( IN := TRUE, PT := T#2s);  (*Start a timer to poll for the accepted connection*)
		IF fbAcceptTON.Q THEN
			fbAcceptTON( IN := FALSE );	(*Reset timer*)
			fb_accept(  bExecute := FALSE  ); (*Generate a rising edge to activate the accept function*)
			fb_accept(hListener := socketHandle, bExecute:= TRUE, hSocket=>activeSocketHandle );
			state:=3; (*Move to the state where the client is accepted*)

			fbAcceptTON( IN := FALSE);

		END_IF
3:
(*Complete accpeting the client connection*)
	fb_accept( bExecute := FALSE ); (*Reset the accept function to try connection again if necessary*)
	IF NOT fb_accept.bBusy THEN
		IF NOT fb_accept.bError THEN
			IF fb_accept.bAccepted THEN
				bAccepted := TRUE; (*If the client connection is accepted without error then move to the send state*)
				fb_accept(bExecute:=FALSE);
				socketToUse:=fb_accept.hSocket;

				state:=4;
			ELSE
				fb_listen(bExecute:=FALSE);
				fb_accept(bExecute:=FALSE);
				arduinoConnected:=FALSE; (*If the connection attempt was not successful, return the boolean as false*)
				fbAcceptTON( IN := FALSE);
				state:=2;

				END_IF
		END_IF
	END_IF
4:
arduinoConnected:=TRUE;
RETURN;

END_CASE;
END_FUNCTION_BLOCK

(* POU ArduinoDisconnect, ST *)
FUNCTION_BLOCK ArduinoDisconnect
VAR_INPUT
	bCloseAll: BOOL;
END_VAR
VAR_OUTPUT
	connectionClosed: BOOL;
END_VAR
VAR
	fb_closeAll: FB_SocketCloseAll;
END_VAR
(*This function closes the TCP/IP port being used the Arduino connection*)

IF bCloseAll THEN
	bCloseAll:=FALSE;
	(*Close all open ports*)
	fb_closeAll(sSrvNetId:='', bExecute:=TRUE, tTimeOut:=T#5s );
ELSE
	fb_closeAll(bExecute:=FALSE);
END_IF


(*Move to the listening state*)
IF NOT fb_closeAll.bError THEN
	connectionClosed:=TRUE;


ELSE
connectionClosed:=FALSE;
END_IF
RETURN;
END_FUNCTION_BLOCK

(* POU ArduinoReceiveData, ST *)
FUNCTION_BLOCK ArduinoReceiveData
VAR_INPUT
	socketToUse: T_HSOCKET;
END_VAR
VAR_OUTPUT
	dataReceived: BOOL;
	heading: LREAL;
	xAccel: LREAL;
	yAccel: LREAL;
END_VAR
VAR
	(*Connection timers*)
	fbReceiveTON: TON;

 	(*Functions*)
	fb_receive: FB_SocketReceive;

	(*Send and receive data and variables*)
	receiveBuffer: ARRAY[0..17] OF BYTE;
	bytesReceived: UDINT;
	sendBuffer: STRING;
	sendBufferAddress: DWORD;
	cbReceived, startPos, endPos, idx : UDINT;
	cbFrame: UDINT;
	sFromClient: T_MaxString;
	overflow: BOOL;
	endFound: BOOL;

	(*Error variables*)
	acceptError: UDINT;
	receiveError: UDINT;

	state: INT:=1;
	yDistString: STRING;
	xDistString: STRING;
	zDistString: STRING;
	headingString: STRING;
	timerOn: BOOL;
	timeUp: BOOL;
	fbresetTON: TON;
END_VAR
CASE state OF
1:
(*Receive information*)
	fbReceiveTON(  IN := FALSE, PT:=T#0s); (*Receive first request immediately*)
	fbReceiveTON(  IN := TRUE ); (*Start a timer to ensure complete transfer of information*)

		IF fbReceiveTON.Q THEN
			fbReceiveTON(  IN := FALSE);
			fb_receive(bExecute:=FALSE);  (*Generate a rising edge to start receiving data*)
			fb_receive
			(
				sSrvNetId:='',
				hSocket :=socketToUse,
				cbLen:=SIZEOF(receiveBuffer)-cbReceived,
				pDest:=ADR(receiveBuffer)+cbReceived,
				tTimeout:=T#5s,
				nRecBytes=>bytesReceived,
				nErrId=>receiveError,
				bExecute:=TRUE,
			);

	(*Move to the receive completion state*)
	state:=2;
	END_IF

2:
(*Continue receiving data*)
	fb_receive( bExecute := FALSE );
	IF NOT fb_receive.bBusy THEN
		IF NOT fb_receive.bError THEN (*If no error has occurred then start the actual receiving of data*)

			IF (fb_receive.nRecBytes>0) THEN (*Bytes have been received*)

				startPos:=cbReceived; (*index of first data byte*)
				endPos:=cbReceived+fb_receive.nRecBytes-1; (*index of last byte*)
				cbReceived:=cbReceived+fb_receive.nRecBytes; (*Calculating the number of received data bytes*)
				cbFrame:=0; (*Reset the frame length*)


				IF cbReceived<SIZEOF(sFromClient) THEN (*no overflow*)
					fbReceiveTON(IN:=FALSE, PT:=T#0S);

					(*Search for the string delimiter(separation character for different strings)*)
					FOR idx:=startPos TO endPos BY 1 DO
						IF receiveBuffer[idx]=0 THEN (*String delimiter found*)
							cbFrame:=idx+1;(*calculate length of received string*)
							MEMCPY(ADR(sFromClient), ADR(receiveBuffer),cbFrame); (*copy the received string to the output variable*)
							MEMMOVE(ADR(receiveBuffer), ADR(receiveBuffer[cbFrame]), cbReceived-cbFrame);(*move remaining data bytes*)
							dataReceived:=TRUE;  	(*Send an acknowledgement of data received*)
							state:=3; (*Move to the receive completion state*)
							endFound:=TRUE;
							EXIT;
						END_IF
					END_FOR
				ELSE(*no more free buffer space-overflow*)

					dataReceived:=FALSE; (*Go to error state*)
					overflow:=TRUE;
					state:=4;
				END_IF
			ELSE(*no data received*)
					fbReceiveTON(IN:=FALSE, PT:=T#1ms);
					state:=1;
			END_IF
		ELSE(*error receiving data, exit function*)
			state:=4;
			dataReceived:=FALSE;
		END_IF
	END_IF

3:
	(*State used to process data*)
	xAccel:=(STRING_TO_LREAL(MID(sFromClient, 7, 1)))/1000;  (*Extract the x distance*)
	yAccel:=(STRING_TO_LREAL(MID(sFromClient, 7, 8)))/1000;
	heading:=(STRING_TO_LREAL(MID(sFromClient, 4, 15)))/10;

	fb_receive(bExecute:=FALSE); (*Reset the receive function*)
	startPos:=0; (*reset buffer beginning pointer*)
	endPos:=0;  (*reset buffer end pointer*)
	cbReceived:=0; (*reset bytes received counter*)
	sFromClient:=''; (*reset transition variable*)


	state:=1;
	RETURN;

4: (*Unused except for as an error state*)
reset:=TRUE;

	(*Clear buffer-PROBABLY UNNECESSARY*)

	receiveBuffer[0]:=0;
	receiveBuffer[1]:=0;
	receiveBuffer[2]:=0;
	receiveBuffer[3]:=0;
	receiveBuffer[4]:=0;
	receiveBuffer[5]:=0;
	receiveBuffer[6]:=0;
	receiveBuffer[7]:=0;
	receiveBuffer[8]:=0;
	receiveBuffer[9]:=0;
	receiveBuffer[10]:=0;
	receiveBuffer[11]:=0;
	receiveBuffer[12]:=0;
	receiveBuffer[13]:=0;
	receiveBuffer[14]:=0;
	receiveBuffer[15]:=0;
receiveBuffer[16]:=0;
receiveBuffer[17]:=0;



	state:=1;


END_CASE;
END_FUNCTION_BLOCK

(* Visualisation MAINGUI
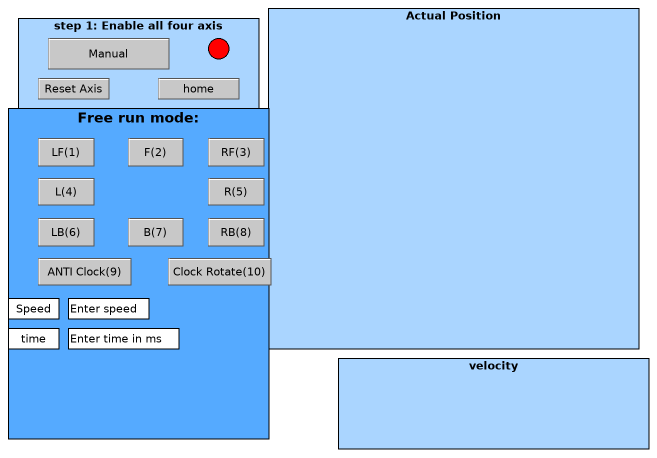
rectangle at (10,20)-(251,121): text "step 1: Enable all four axis"
button at (40,40)-(161,71): text "Manual"; toggles MAIN.Manual
ellipse at (200,40)-(221,61): alarm colour if .trigger2
button at (30,80)-(101,101): text "Reset Axis"; taps reset
rectangle at (260,10)-(631,351): text "Actual Position"
rectangle at (0,110)-(261,441): text "Free run mode:"
button at (30,140)-(86,168): text "LF(1)"; taps MAIN.bMoveCombination[1]
button at (30,180)-(86,207): text "L(4)"; taps MAIN.bMoveCombination[4]
button at (30,220)-(86,248): text "LB(6)"; taps MAIN.bMoveCombination[6]
button at (120,140)-(175,168): text "F(2)"; taps MAIN.bMoveCombination[2]
button at (120,220)-(175,248): text "B(7)"; taps MAIN.bMoveCombination[7]
button at (200,140)-(256,168): text "RF(3)"; taps MAIN.bMoveCombination[3]
button at (200,180)-(256,207): text "R(5)"; taps MAIN.bMoveCombination[5]
button at (200,220)-(256,248): text "RB(8)"; taps MAIN.bMoveCombination[8]
button at (30,260)-(123,287): text "ANTI Clock(9)"; taps MAIN.bMoveCombination[9]
button at (160,260)-(263,287): text "Clock Rotate(10)"; taps MAIN.bMoveCombination[10]
rectangle at (60,330)-(171,351): text "Enter time in ms"; shows MAIN.timeToMoveReal; editable 0..20000
rectangle at (330,360)-(641,451): text "velocity"
rectangle at (60,300)-(141,321): text "Enter speed"; shows MAIN.speedToMove; editable 0..2000
rectangle at (0,330)-(51,351): text "time"
rectangle at (0,300)-(51,321): text "Speed"
button at (150,80)-(231,101): text "home"; taps home
21 elements of other kinds (tables, trends, ...) not read
*)
